LIN {X 0,Y 382.688,Z 736.187,A -85,B 0,C 180,E1 16955.399,E2 16955.399} C_VEL
LIN {X 0,Y 386.297,Z 719.198,A -85,B 0,C 180,E1 16953.634,E2 16953.634} C_VEL
LIN {X 0,Y 389.635,Z 701.414,A -85,B 0,C 180,E1 16952.136,E2 16952.136} C_VEL
LIN {X 0,Y 392.651,Z 682.888,A -85,B 0,C 180,E1 16950.895,E2 16950.895} C_VEL
LIN {X 0,Y 395.335,Z 662.731,A -85,B 0,C 180,E1 16949.855,E2 16949.855} C_VEL
LIN {X 0,Y 397.472,Z 642.044,A -85,B 0,C 180,E1 16949.087,E2 16949.087} C_VEL
LIN {X 0,Y 399.251,Z 615.615,A -85,B 0,C 180,E1 16948.447,E2 16948.447} C_VEL
LIN {X 0,Y 408.41,Z 452.206,A -85,B 0,C 180,E1 16945.014,E2 16945.014} C_VEL
LIN {X 0,Y 404.369,Z 398.592,A -85,B 0,C 180,E1 16942.698,E2 16942.698} C_VEL
LIN {X 0,Y 403.693,Z 388.775,A -85,B 0,C 180,E1 16942.223,E2 16942.223} C_VEL
LIN {X 0,Y 411.245,Z 343.049,A -85,B 0,C 180,E1 16938.531,E2 16938.531} C_VEL
LIN {X 0,Y 405.242,Z 328.597,A -85,B 0,C 180,E1 16935.6,E2 16935.6} C_VEL
LIN {X 0,Y 399.503,Z 315.936,A -85,B 0,C 180,E1 16932.576,E2 16932.576} C_VEL
LIN {X 0,Y 394.557,Z 306.307,A -85,B 0,C 180,E1 16929.775,E2 16929.775} C_VEL
LIN {X 0,Y 390.908,Z 299.036,A -85,B 0,C 180,E1 16927.347,E2 16927.347} C_VEL
LIN {X 0,Y 387.906,Z 293.83,A -85,B 0,C 180,E1 16925.175,E2 16925.175} C_VEL
LIN {X 0,Y 385.327,Z 289.182,A -85,B 0,C 180,E1 16922.974,E2 16922.974} C_VEL
LIN {X 0,Y 382.942,Z 284.925,A -85,B 0,C 180,E1 16920.436,E2 16920.436} C_VEL
LIN {X 0,Y 382.29,Z 283.961,A -85,B 0,C 180,E1 16919.7,E2 16919.7} C_VEL
LIN {X 0,Y 379.591,Z 279.036,A -85,B 0,C 180,E1 16914.407,E2 16914.407} C_VEL
LIN {X 0,Y 379.173,Z 278.59,A -85,B 0,C 180,E1 16910.59,E2 16910.59} C_VEL
LIN {X 0,Y 379.911,Z 279.467,A -85,B 0,C 180,E1 16907.691,E2 16907.691} C_VEL
LIN {X 0,Y 382.64,Z 284.104,A -85,B 0,C 180,E1 16903.139,E2 16903.139} C_VEL
LIN {X 0,Y 383.425,Z 284.941,A -85,B 0,C 180,E1 16902.392,E2 16902.392} C_VEL
LIN {X 0,Y 385.824,Z 289.277,A -85,B 0,C 180,E1 16899.996,E2 16899.996} C_VEL
LIN {X 0,Y 386.815,Z 290.588,A -85,B 0,C 180,E1 16899.26,E2 16899.26} C_VEL
LIN {X 0,Y 389.166,Z 294.616,A -85,B 0,C 180,E1 16897.491,E2 16897.491} C_VEL
LIN {X 0,Y 393.023,Z 301.294,A -85,B 0,C 180,E1 16895.019,E2 16895.019} C_VEL
LIN {X 0,Y 397.476,Z 309.022,A -85,B 0,C 180,E1 16892.591,E2 16892.591} C_VEL
LIN {X 0,Y 402.971,Z 319.612,A -85,B 0,C 180,E1 16889.92,E2 16889.92} C_VEL
LIN {X 0,Y 408.692,Z 331.236,A -85,B 0,C 180,E1 16887.437,E2 16887.437} C_VEL
LIN {X 0,Y 411.334,Z 336.632,A -85,B 0,C 180,E1 16886.468,E2 16886.468} C_VEL
LIN {X 0,Y 417.132,Z 345.96,A -85,B 0,C 180,E1 16885.268,E2 16885.268} C_VEL
LIN {X 0,Y 417.545,Z 355.442,A -85,B 0,C 180,E1 16884.962,E2 16884.962} C_VEL
LIN {X 0,Y 410.945,Z 542.625,A -85,B 0,C 180,E1 16881.466,E2 16881.466} C_VEL
LIN {X 0,Y 407.268,Z 659.162,A -85,B 0,C 180,E1 16879.351,E2 16879.351} C_VEL
LIN {X 0,Y 405.386,Z 681.756,A -85,B 0,C 180,E1 16878.737,E2 16878.737} C_VEL
LIN {X 0,Y 402.869,Z 703.945,A -85,B 0,C 180,E1 16877.905,E2 16877.905} C_VEL
LIN {X 0,Y 399.919,Z 724.711,A -85,B 0,C 180,E1 16876.887,E2 16876.887} C_VEL
LIN {X 0,Y 396.281,Z 746.248,A -85,B 0,C 180,E1 16875.562,E2 16875.562} C_VEL
LIN {X 0,Y 392.531,Z 766.4,A -85,B 0,C 180,E1 16874.055,E2 16874.055} C_VEL
LIN {X 0,Y 388.456,Z 785.774,A -85,B 0,C 180,E1 16872.303,E2 16872.303} C_VEL
LIN {X 0,Y 384.097,Z 805.442,A -85,B 0,C 180,E1 16870.207,E2 16870.207} C_VEL
LIN {X 0,Y 380.023,Z 823.04,A -85,B 0,C 180,E1 16867.998,E2 16867.998} C_VEL
LIN {X 0,Y 375.819,Z 840.992,A -85,B 0,C 180,E1 16865.353,E2 16865.353} C_VEL
LIN {X 0,Y 372.203,Z 856.686,A -85,B 0,C 180,E1 16862.678,E2 16862.678} C_VEL
LIN {X 0,Y 368.937,Z 871.382,A -85,B 0,C 180,E1 16859.73,E2 16859.73} C_VEL
LIN {X 0,Y 366.041,Z 885.503,A -85,B 0,C 180,E1 16856.437,E2 16856.437} C_VEL
LIN {X 0,Y 363.942,Z 896.95,A -85,B 0,C 180,E1 16853.302,E2 16853.302} C_VEL
LIN {X 0,Y 362.3,Z 907.595,A -85,B 0,C 180,E1 16849.841,E2 16849.841} C_VEL
LIN {X 0,Y 361.331,Z 915.623,A -85,B 0,C 180,E1 16846.723,E2 16846.723} C_VEL
LIN {X 0,Y 360.676,Z 923.062,A -85,B 0,C 180,E1 16843.137,E2 16843.137} C_VEL
LIN {X 0,Y 360.397,Z 928.023,A -85,B 0,C 180,E1 16840.064,E2 16840.064} C_VEL
LIN {X 0,Y 360.333,Z 932.128,A -85,B 0,C 180,E1 16836.531,E2 16836.531} C_VEL
LIN {X 0,Y 360.329,Z 934.234,A -85,B 0,C 180,E1 16833.498,E2 16833.498} C_VEL
LIN {X 0,Y 360.326,Z 935.127,A -85,B 0,C 180,E1 16830.475,E2 16830.475} C_VEL
LIN {X 0,Y 360.322,Z 934.598,A -85,B 0,C 180,E1 16827.135,E2 16827.135} C_VEL
LIN {X 0,Y 360.305,Z 932.768,A -85,B 0,C 180,E1 16824.105,E2 16824.105} C_VEL
LIN {X 0,Y 360.331,Z 929.542,A -85,B 0,C 180,E1 16820.898,E2 16820.898} C_VEL
LIN {X 0,Y 360.586,Z 924.375,A -85,B 0,C 180,E1 16817.435,E2 16817.435} C_VEL
LIN {X 0,Y 361.071,Z 918.244,A -85,B 0,C 180,E1 16814.252,E2 16814.252} C_VEL
LIN {X 0,Y 362.037,Z 909.95,A -85,B 0,C 180,E1 16810.812,E2 16810.812} C_VEL
LIN {X 0,Y 363.482,Z 900.51,A -85,B 0,C 180,E1 16807.558,E2 16807.558} C_VEL
LIN {X 0,Y 365.577,Z 888.949,A -85,B 0,C 180,E1 16804.222,E2 16804.222} C_VEL
LIN {X 0,Y 368.207,Z 876.331,A -85,B 0,C 180,E1 16801.094,E2 16801.094} C_VEL
LIN {X 0,Y 371.344,Z 862.246,A -85,B 0,C 180,E1 16798.146,E2 16798.146} C_VEL
LIN {X 0,Y 375.147,Z 846.088,A -85,B 0,C 180,E1 16795.223,E2 16795.223} C_VEL
LIN {X 0,Y 379.148,Z 829.472,A -85,B 0,C 180,E1 16792.659,E2 16792.659} C_VEL
LIN {X 0,Y 383.39,Z 811.434,A -85,B 0,C 180,E1 16790.285,E2 16790.285} C_VEL
LIN {X 0,Y 387.72,Z 792.747,A -85,B 0,C 180,E1 16788.183,E2 16788.183} C_VEL
LIN {X 0,Y 391.873,Z 773.311,A -85,B 0,C 180,E1 16786.354,E2 16786.354} C_VEL
LIN {X 0,Y 396.014,Z 752.373,A -85,B 0,C 180,E1 16784.697,E2 16784.697} C_VEL
LIN {X 0,Y 399.383,Z 733.203,A -85,B 0,C 180,E1 16783.445,E2 16783.445} C_VEL
LIN {X 0,Y 402.81,Z 710.278,A -85,B 0,C 180,E1 16782.24,E2 16782.24} C_VEL
LIN {X 0,Y 405.545,Z 688.092,A -85,B 0,C 180,E1 16781.334,E2 16781.334} C_VEL
LIN {X 0,Y 407.597,Z 665.402,A -85,B 0,C 180,E1 16780.677,E2 16780.677} C_VEL
LIN {X 0,Y 408.984,Z 634.84,A -85,B 0,C 180,E1 16780.061,E2 16780.061} C_VEL
LIN {X 0,Y 415.34,Z 444.739,A -85,B 0,C 180,E1 16776.571,E2 16776.571} C_VEL
LIN {X 0,Y 418.612,Z 352.233,A -85,B 0,C 180,E1 16774.81,E2 16774.81} C_VEL
LIN {X 0,Y 418.047,Z 346.712,A -85,B 0,C 180,E1 16774.593,E2 16774.593} C_VEL
LIN {X 0,Y 406.732,Z 329.749,A -85,B 0,C 180,E1 16772.405,E2 16772.405} C_VEL
LIN {X 0,Y 397.743,Z 312.998,A -85,B 0,C 180,E1 16769.189,E2 16769.189} C_VEL
LIN {X 0,Y 388.439,Z 296.63,A -85,B 0,C 180,E1 16765.541,E2 16765.541} C_VEL
LIN {X 0,Y 381.638,Z 285.645,A -85,B 0,C 180,E1 16762.652,E2 16762.652} C_VEL
LIN {X 0,Y 378.529,Z 280.582,A -85,B 0,C 180,E1 16761.216,E2 16761.216} C_VEL
LIN {X 0,Y 375.523,Z 275.76,A -85,B 0,C 180,E1 16759.764,E2 16759.764} C_VEL
LIN {X 0,Y 372.969,Z 271.522,A -85,B 0,C 180,E1 16758.442,E2 16758.442} C_VEL
LIN {X 0,Y 369.781,Z 266.966,A -85,B 0,C 180,E1 16756.818,E2 16756.818} C_VEL
LIN {X 0,Y 369.096,Z 265.429,A -85,B 0,C 180,E1 16756.364,E2 16756.364} C_VEL
LIN {X 0,Y 366.486,Z 262.302,A -85,B 0,C 180,E1 16755.022,E2 16755.022} C_VEL
LIN {X 0,Y 365.135,Z 259.526,A -85,B 0,C 180,E1 16754.106,E2 16754.106} C_VEL
LIN {X 0,Y 362.664,Z 256.791,A -85,B 0,C 180,E1 16752.742,E2 16752.742} C_VEL
LIN {X 0,Y 361.846,Z 254.324,A -85,B 0,C 180,E1 16751.88,E2 16751.88} C_VEL
LIN {X 0,Y 361.788,Z 253.955,A -85,B 0,C 180,E1 16749.706,E2 16749.706} C_VEL
LIN {X 0,Y 361.798,Z 253.95,A -85,B 0,C 180,E1 16745.71,E2 16745.71} C_VEL
LIN {X 0,Y 361.799,Z 253.95,A -85,B 0,C 180,E1 16741.584,E2 16741.584} C_VEL
LIN {X 0,Y 361.798,Z 253.959,A -85,B 0,C 180,E1 16737.466,E2 16737.466} C_VEL
LIN {X 0,Y 361.808,Z 253.977,A -85,B 0,C 180,E1 16733.335,E2 16733.335} C_VEL
LIN {X 0,Y 361.798,Z 253.972,A -85,B 0,C 180,E1 16729.169,E2 16729.169} C_VEL
LIN {X 0,Y 361.807,Z 253.951,A -85,B 0,C 180,E1 16725.108,E2 16725.108} C_VEL
LIN {X 0,Y 361.801,Z 253.946,A -85,B 0,C 180,E1 16720.936,E2 16720.936} C_VEL
LIN {X 0,Y 361.808,Z 253.959,A -85,B 0,C 180,E1 16716.896,E2 16716.896} C_VEL
LIN {X 0,Y 361.807,Z 253.98,A -85,B 0,C 180,E1 16712.695,E2 16712.695} C_VEL
LIN {X 0,Y 361.804,Z 253.97,A -85,B 0,C 180,E1 16708.514,E2 16708.514} C_VEL
LIN {X 0,Y 361.798,Z 253.956,A -85,B 0,C 180,E1 16704.331,E2 16704.331} C_VEL
LIN {X 0,Y 361.801,Z 253.949,A -85,B 0,C 180,E1 16700.2,E2 16700.2} C_VEL
LIN {X 0,Y 361.8,Z 253.95,A -85,B 0,C 180,E1 16696.081,E2 16696.081} C_VEL
LIN {X 0,Y 361.802,Z 253.953,A -85,B 0,C 180,E1 16691.975,E2 16691.975} C_VEL
LIN {X 0,Y 361.843,Z 254.237,A -85,B 0,C 180,E1 16690.381,E2 16690.381} C_VEL
LIN {X 0,Y 363.417,Z 257.875,A -85,B 0,C 180,E1 16689.055,E2 16689.055} C_VEL
LIN {X 0,Y 365.534,Z 260.297,A -85,B 0,C 180,E1 16687.896,E2 16687.896} C_VEL
LIN {X 0,Y 367.518,Z 264.005,A -85,B 0,C 180,E1 16686.626,E2 16686.626} C_VEL
LIN {X 0,Y 368.956,Z 265.786,A -85,B 0,C 180,E1 16685.878,E2 16685.878} C_VEL
LIN {X 0,Y 371.04,Z 269.542,A -85,B 0,C 180,E1 16684.653,E2 16684.653} C_VEL
LIN {X 0,Y 372.261,Z 271.21,A -85,B 0,C 180,E1 16684.046,E2 16684.046} C_VEL
LIN {X 0,Y 374.624,Z 275.216,A -85,B 0,C 180,E1 16682.785,E2 16682.785} C_VEL
LIN {X 0,Y 378.879,Z 282.66,A -85,B 0,C 180,E1 16680.62,E2 16680.62} C_VEL
LIN {X 0,Y 383.531,Z 290.759,A -85,B 0,C 180,E1 16678.42,E2 16678.42} C_VEL
LIN {X 0,Y 390.609,Z 304.107,A -85,B 0,C 180,E1 16675.236,E2 16675.236} C_VEL
LIN {X 0,Y 397.071,Z 317.353,A -85,B 0,C 180,E1 16672.464,E2 16672.464} C_VEL
LIN {X 0,Y 403.782,Z 332.36,A -85,B 0,C 180,E1 16669.681,E2 16669.681} C_VEL
LIN {X 0,Y 405.757,Z 337.501,A -85,B 0,C 180,E1 16668.834,E2 16668.834} C_VEL
LIN {X 0,Y 398.051,Z 391.605,A -85,B 0,C 180,E1 16664.549,E2 16664.549} C_VEL
LIN {X 0,Y 397.459,Z 397.862,A -85,B 0,C 180,E1 16664.105,E2 16664.105} C_VEL
LIN {X 0,Y 402.131,Z 451.79,A -85,B 0,C 180,E1 16662.007,E2 16662.007} C_VEL
LIN {X 0,Y 393.972,Z 628.533,A -85,B 0,C 180,E1 16658.434,E2 16658.434} C_VEL
LIN {X 0,Y 392.449,Z 649.279,A -85,B 0,C 180,E1 16657.835,E2 16657.835} C_VEL
LIN {X 0,Y 391.777,Z 656.525,A -85,B 0,C 180,E1 16657.565,E2 16657.565} C_VEL
LIN {X 0,Y 390.077,Z 664.06,A -85,B 0,C 180,E1 16657.353,E2 16657.353} C_VEL
LIN {X 0,Y 383.174,Z 682.726,A -85,B 0,C 180,E1 16656.918,E2 16656.918} C_VEL
LIN {X 0,Y 381.385,Z 689.741,A -85,B 0,C 180,E1 16656.564,E2 16656.564} C_VEL
LIN {X 0,Y 378.3,Z 708.589,A -85,B 0,C 180,E1 16655.157,E2 16655.157} C_VEL
LIN {X 0,Y 375.005,Z 726.153,A -85,B 0,C 180,E1 16653.517,E2 16653.517} C_VEL
LIN {X 0,Y 371.571,Z 742.681,A -85,B 0,C 180,E1 16651.621,E2 16651.621} C_VEL
LIN {X 0,Y 368.244,Z 757.61,A -85,B 0,C 180,E1 16649.535,E2 16649.535} C_VEL
LIN {X 0,Y 364.986,Z 771.54,A -85,B 0,C 180,E1 16647.175,E2 16647.175} C_VEL
LIN {X 0,Y 362.021,Z 783.964,A -85,B 0,C 180,E1 16644.613,E2 16644.613} C_VEL
LIN {X 0,Y 359.452,Z 794.899,A -85,B 0,C 180,E1 16641.846,E2 16641.846} C_VEL
LIN {X 0,Y 357.411,Z 803.86,A -85,B 0,C 180,E1 16639.036,E2 16639.036} C_VEL
LIN {X 0,Y 355.833,Z 811.436,A -85,B 0,C 180,E1 16636.018,E2 16636.018} C_VEL
LIN {X 0,Y 354.721,Z 817.412,A -85,B 0,C 180,E1 16632.848,E2 16632.848} C_VEL
LIN {X 0,Y 354.064,Z 821.587,A -85,B 0,C 180,E1 16629.641,E2 16629.641} C_VEL
LIN {X 0,Y 353.771,Z 823.967,A -85,B 0,C 180,E1 16626.517,E2 16626.517} C_VEL
LIN {X 0,Y 353.745,Z 824.748,A -85,B 0,C 180,E1 16623.272,E2 16623.272} C_VEL
LIN {X 0,Y 353.963,Z 823.882,A -85,B 0,C 180,E1 16620.133,E2 16620.133} C_VEL
LIN {X 0,Y 354.483,Z 821.421,A -85,B 0,C 180,E1 16617.02,E2 16617.02} C_VEL
LIN {X 0,Y 355.382,Z 817.422,A -85,B 0,C 180,E1 16613.986,E2 16613.986} C_VEL
LIN {X 0,Y 356.758,Z 811.625,A -85,B 0,C 180,E1 16610.909,E2 16610.909} C_VEL
LIN {X 0,Y 358.765,Z 803.801,A -85,B 0,C 180,E1 16607.808,E2 16607.808} C_VEL
LIN {X 0,Y 361.316,Z 794.333,A -85,B 0,C 180,E1 16604.881,E2 16604.881} C_VEL
LIN {X 0,Y 364.284,Z 783.463,A -85,B 0,C 180,E1 16602.18,E2 16602.18} C_VEL
LIN {X 0,Y 367.641,Z 771.125,A -85,B 0,C 180,E1 16599.68,E2 16599.68} C_VEL
LIN {X 0,Y 371.24,Z 757.424,A -85,B 0,C 180,E1 16597.393,E2 16597.393} C_VEL
LIN {X 0,Y 375.158,Z 741.609,A -85,B 0,C 180,E1 16595.231,E2 16595.231} C_VEL
LIN {X 0,Y 378.942,Z 725.002,A -85,B 0,C 180,E1 16593.378,E2 16593.378} C_VEL
LIN {X 0,Y 382.663,Z 706.838,A -85,B 0,C 180,E1 16591.738,E2 16591.738} C_VEL
LIN {X 0,Y 385.974,Z 688.136,A -85,B 0,C 180,E1 16590.391,E2 16590.391} C_VEL
LIN {X 0,Y 388.913,Z 668.177,A -85,B 0,C 180,E1 16589.28,E2 16589.28} C_VEL
LIN {X 0,Y 391.268,Z 647.69,A -85,B 0,C 180,E1 16588.442,E2 16588.442} C_VEL
LIN {X 0,Y 392.994,Z 626.19,A -85,B 0,C 180,E1 16587.852,E2 16587.852} C_VEL
LIN {X 0,Y 403.129,Z 453.659,A -85,B 0,C 180,E1 16584.186,E2 16584.186} C_VEL
LIN {X 0,Y 399.359,Z 400.422,A -85,B 0,C 180,E1 16581.845,E2 16581.845} C_VEL
LIN {X 0,Y 398.52,Z 387.636,A -85,B 0,C 180,E1 16581.217,E2 16581.217} C_VEL
LIN {X 0,Y 405.502,Z 347.225,A -85,B 0,C 180,E1 16577.914,E2 16577.914} C_VEL
LIN {X 0,Y 399.966,Z 333.564,A -85,B 0,C 180,E1 16575.069,E2 16575.069} C_VEL
LIN {X 0,Y 394.644,Z 321.669,A -85,B 0,C 180,E1 16572.138,E2 16572.138} C_VEL
LIN {X 0,Y 389.914,Z 312.135,A -85,B 0,C 180,E1 16569.296,E2 16569.296} C_VEL
LIN {X 0,Y 386.341,Z 305.126,A -85,B 0,C 180,E1 16566.837,E2 16566.837} C_VEL
LIN {X 0,Y 383.92,Z 300.595,A -85,B 0,C 180,E1 16564.93,E2 16564.93} C_VEL
LIN {X 0,Y 381.583,Z 296.206,A -85,B 0,C 180,E1 16562.853,E2 16562.853} C_VEL
LIN {X 0,Y 379.28,Z 292.042,A -85,B 0,C 180,E1 16560.302,E2 16560.302} C_VEL
LIN {X 0,Y 378.639,Z 291.04,A -85,B 0,C 180,E1 16559.546,E2 16559.546} C_VEL
LIN {X 0,Y 376.196,Z 286.275,A -85,B 0,C 180,E1 16554.356,E2 16554.356} C_VEL
LIN {X 0,Y 375.815,Z 285.853,A -85,B 0,C 180,E1 16550.66,E2 16550.66} C_VEL
LIN {X 0,Y 376.492,Z 286.609,A -85,B 0,C 180,E1 16547.889,E2 16547.889} C_VEL
LIN {X 0,Y 379.308,Z 291.4,A -85,B 0,C 180,E1 16543.104,E2 16543.104} C_VEL
LIN {X 0,Y 379.969,Z 292.424,A -85,B 0,C 180,E1 16542.385,E2 16542.385} C_VEL
LIN {X 0,Y 382.656,Z 296.799,A -85,B 0,C 180,E1 16539.823,E2 16539.823} C_VEL
LIN {X 0,Y 386.131,Z 302.923,A -85,B 0,C 180,E1 16537.144,E2 16537.144} C_VEL
LIN {X 0,Y 389.061,Z 308.123,A -85,B 0,C 180,E1 16535.235,E2 16535.235} C_VEL
LIN {X 0,Y 393.424,Z 315.935,A -85,B 0,C 180,E1 16532.777,E2 16532.777} C_VEL
LIN {X 0,Y 398.532,Z 325.948,A -85,B 0,C 180,E1 16530.214,E2 16530.214} C_VEL
LIN {X 0,Y 404.028,Z 337.304,A -85,B 0,C 180,E1 16527.771,E2 16527.771} C_VEL
LIN {X 0,Y 412.063,Z 350.006,A -85,B 0,C 180,E1 16525.992,E2 16525.992} C_VEL
LIN {X 0,Y 412.277,Z 356.873,A -85,B 0,C 180,E1 16525.778,E2 16525.778} C_VEL
LIN {X 0,Y 405.196,Z 546.047,A -85,B 0,C 180,E1 16522.205,E2 16522.205} C_VEL
LIN {X 0,Y 401.455,Z 658.643,A -85,B 0,C 180,E1 16520.14,E2 16520.14} C_VEL
LIN {X 0,Y 399.525,Z 681.093,A -85,B 0,C 180,E1 16519.526,E2 16519.526} C_VEL
LIN {X 0,Y 396.954,Z 702.973,A -85,B 0,C 180,E1 16518.705,E2 16518.705} C_VEL
LIN {X 0,Y 393.979,Z 723.237,A -85,B 0,C 180,E1 16517.71,E2 16517.71} C_VEL
LIN {X 0,Y 390.175,Z 744.944,A -85,B 0,C 180,E1 16516.377,E2 16516.377} C_VEL
LIN {X 0,Y 386.094,Z 765.857,A -85,B 0,C 180,E1 16514.8,E2 16514.8} C_VEL
LIN {X 0,Y 381.823,Z 785.265,A -85,B 0,C 180,E1 16513.02,E2 16513.02} C_VEL
LIN {X 0,Y 377.134,Z 805.454,A -85,B 0,C 180,E1 16510.826,E2 16510.826} C_VEL
LIN {X 0,Y 372.713,Z 823.659,A -85,B 0,C 180,E1 16508.487,E2 16508.487} C_VEL
LIN {X 0,Y 368.468,Z 840.841,A -85,B 0,C 180,E1 16505.88,E2 16505.88} C_VEL
LIN {X 0,Y 364.583,Z 856.807,A -85,B 0,C 180,E1 16503.074,E2 16503.074} C_VEL
LIN {X 0,Y 361.194,Z 871.379,A -85,B 0,C 180,E1 16500.067,E2 16500.067} C_VEL
LIN {X 0,Y 358.189,Z 885.306,A -85,B 0,C 180,E1 16496.704,E2 16496.704} C_VEL
LIN {X 0,Y 355.929,Z 897.222,A -85,B 0,C 180,E1 16493.332,E2 16493.332} C_VEL
LIN {X 0,Y 354.338,Z 907.121,A -85,B 0,C 180,E1 16489.962,E2 16489.962} C_VEL
LIN {X 0,Y 353.271,Z 915.827,A -85,B 0,C 180,E1 16486.439,E2 16486.439} C_VEL
LIN {X 0,Y 352.71,Z 922.339,A -85,B 0,C 180,E1 16483.106,E2 16483.106} C_VEL
LIN {X 0,Y 352.438,Z 927.45,A -85,B 0,C 180,E1 16479.799,E2 16479.799} C_VEL
LIN {X 0,Y 352.416,Z 931.153,A -85,B 0,C 180,E1 16476.351,E2 16476.351} C_VEL
LIN {X 0,Y 352.417,Z 933.167,A -85,B 0,C 180,E1 16473.251,E2 16473.251} C_VEL
LIN {X 0,Y 352.426,Z 933.964,A -85,B 0,C 180,E1 16469.836,E2 16469.836} C_VEL
LIN {X 0,Y 352.406,Z 933.164,A -85,B 0,C 180,E1 16466.583,E2 16466.583} C_VEL
LIN {X 0,Y 352.389,Z 931.171,A -85,B 0,C 180,E1 16463.482,E2 16463.482} C_VEL
LIN {X 0,Y 352.428,Z 927.232,A -85,B 0,C 180,E1 16459.868,E2 16459.868} C_VEL
LIN {X 0,Y 352.699,Z 922.401,A -85,B 0,C 180,E1 16456.723,E2 16456.723} C_VEL
LIN {X 0,Y 353.328,Z 915.548,A -85,B 0,C 180,E1 16453.222,E2 16453.222} C_VEL
LIN {X 0,Y 354.392,Z 907.299,A -85,B 0,C 180,E1 16449.865,E2 16449.865} C_VEL
LIN {X 0,Y 356.129,Z 896.907,A -85,B 0,C 180,E1 16446.328,E2 16446.328} C_VEL
LIN {X 0,Y 358.359,Z 885.68,A -85,B 0,C 180,E1 16443.127,E2 16443.127} C_VEL
LIN {X 0,Y 361.444,Z 871.823,A -85,B 0,C 180,E1 16439.769,E2 16439.769} C_VEL
LIN {X 0,Y 365.071,Z 856.773,A -85,B 0,C 180,E1 16436.651,E2 16436.651} C_VEL
LIN {X 0,Y 369.093,Z 840.617,A -85,B 0,C 180,E1 16433.83,E2 16433.83} C_VEL
LIN {X 0,Y 373.575,Z 822.695,A -85,B 0,C 180,E1 16431.156,E2 16431.156} C_VEL
LIN {X 0,Y 378.141,Z 804.314,A -85,B 0,C 180,E1 16428.821,E2 16428.821} C_VEL
LIN {X 0,Y 382.576,Z 785.189,A -85,B 0,C 180,E1 16426.784,E2 16426.784} C_VEL
LIN {X 0,Y 386.861,Z 765.624,A -85,B 0,C 180,E1 16425.018,E2 16425.018} C_VEL
LIN {X 0,Y 390.768,Z 745.695,A -85,B 0,C 180,E1 16423.527,E2 16423.527} C_VEL
LIN {X 0,Y 394.634,Z 723.464,A -85,B 0,C 180,E1 16422.176,E2 16422.176} C_VEL
LIN {X 0,Y 397.727,Z 702.475,A -85,B 0,C 180,E1 16421.154,E2 16421.154} C_VEL
LIN {X 0,Y 400.204,Z 680.919,A -85,B 0,C 180,E1 16420.364,E2 16420.364} C_VEL
LIN {X 0,Y 402.111,Z 658.063,A -85,B 0,C 180,E1 16419.752,E2 16419.752} C_VEL
LIN {X 0,Y 409.524,Z 448.97,A -85,B 0,C 180,E1 16415.862,E2 16415.862} C_VEL
LIN {X 0,Y 413.094,Z 353.38,A -85,B 0,C 180,E1 16414.021,E2 16414.021} C_VEL
LIN {X 0,Y 412.732,Z 350.864,A -85,B 0,C 180,E1 16413.903,E2 16413.903} C_VEL
LIN {X 0,Y 400.038,Z 332.096,A -85,B 0,C 180,E1 16411.408,E2 16411.408} C_VEL
LIN {X 0,Y 391.985,Z 317.207,A -85,B 0,C 180,E1 16408.489,E2 16408.489} C_VEL
LIN {X 0,Y 383.66,Z 302.559,A -85,B 0,C 180,E1 16405.138,E2 16405.138} C_VEL
LIN {X 0,Y 377.067,Z 291.755,A -85,B 0,C 180,E1 16402.264,E2 16402.264} C_VEL
LIN {X 0,Y 373.99,Z 286.758,A -85,B 0,C 180,E1 16400.829,E2 16400.829} C_VEL
LIN {X 0,Y 371.353,Z 282.381,A -85,B 0,C 180,E1 16399.504,E2 16399.504} C_VEL
LIN {X 0,Y 367.881,Z 276.964,A -85,B 0,C 180,E1 16397.723,E2 16397.723} C_VEL
LIN {X 0,Y 365.437,Z 273.053,A -85,B 0,C 180,E1 16396.369,E2 16396.369} C_VEL
LIN {X 0,Y 364.319,Z 271.513,A -85,B 0,C 180,E1 16395.766,E2 16395.766} C_VEL
LIN {X 0,Y 361.953,Z 267.903,A -85,B 0,C 180,E1 16394.396,E2 16394.396} C_VEL
LIN {X 0,Y 361.313,Z 266.486,A -85,B 0,C 180,E1 16393.932,E2 16393.932} C_VEL
LIN {X 0,Y 358.607,Z 263.337,A -85,B 0,C 180,E1 16392.398,E2 16392.398} C_VEL
LIN {X 0,Y 357.402,Z 260.703,A -85,B 0,C 180,E1 16391.457,E2 16391.457} C_VEL
LIN {X 0,Y 354.849,Z 257.921,A -85,B 0,C 180,E1 16389.898,E2 16389.898} C_VEL
LIN {X 0,Y 353.871,Z 255.276,A -85,B 0,C 180,E1 16388.777,E2 16388.777} C_VEL
LIN {X 0,Y 353.856,Z 254.939,A -85,B 0,C 180,E1 16385.676,E2 16385.676} C_VEL
LIN {X 0,Y 353.853,Z 254.938,A -85,B 0,C 180,E1 16381.458,E2 16381.458} C_VEL
LIN {X 0,Y 353.856,Z 254.946,A -85,B 0,C 180,E1 16377.409,E2 16377.409} C_VEL
LIN {X 0,Y 353.858,Z 254.962,A -85,B 0,C 180,E1 16373.185,E2 16373.185} C_VEL
LIN {X 0,Y 353.85,Z 254.966,A -85,B 0,C 180,E1 16368.923,E2 16368.923} C_VEL
LIN {X 0,Y 353.851,Z 254.945,A -85,B 0,C 180,E1 16364.765,E2 16364.765} C_VEL
LIN {X 0,Y 353.852,Z 254.935,A -85,B 0,C 180,E1 16360.696,E2 16360.696} C_VEL
LIN {X 0,Y 353.855,Z 254.942,A -85,B 0,C 180,E1 16356.522,E2 16356.522} C_VEL
LIN {X 0,Y 353.858,Z 254.963,A -85,B 0,C 180,E1 16352.394,E2 16352.394} C_VEL
LIN {X 0,Y 353.86,Z 254.964,A -85,B 0,C 180,E1 16348.268,E2 16348.268} C_VEL
LIN {X 0,Y 353.857,Z 254.948,A -85,B 0,C 180,E1 16344.005,E2 16344.005} C_VEL
LIN {X 0,Y 353.857,Z 254.941,A -85,B 0,C 180,E1 16339.723,E2 16339.723} C_VEL
LIN {X 0,Y 353.86,Z 254.938,A -85,B 0,C 180,E1 16335.515,E2 16335.515} C_VEL
LIN {X 0,Y 353.907,Z 255.258,A -85,B 0,C 180,E1 16333.357,E2 16333.357} C_VEL
LIN {X 0,Y 355.515,Z 258.902,A -85,B 0,C 180,E1 16331.803,E2 16331.803} C_VEL
LIN {X 0,Y 357.682,Z 261.181,A -85,B 0,C 180,E1 16330.507,E2 16330.507} C_VEL
LIN {X 0,Y 359.243,Z 264.517,A -85,B 0,C 180,E1 16329.311,E2 16329.311} C_VEL
LIN {X 0,Y 361.241,Z 266.855,A -85,B 0,C 180,E1 16328.182,E2 16328.182} C_VEL
LIN {X 0,Y 363.371,Z 270.753,A -85,B 0,C 180,E1 16326.803,E2 16326.803} C_VEL
LIN {X 0,Y 364.633,Z 272.426,A -85,B 0,C 180,E1 16326.127,E2 16326.127} C_VEL
LIN {X 0,Y 367.156,Z 276.625,A -85,B 0,C 180,E1 16324.674,E2 16324.674} C_VEL
LIN {X 0,Y 371.11,Z 283.453,A -85,B 0,C 180,E1 16322.512,E2 16322.512} C_VEL
LIN {X 0,Y 374.333,Z 289.087,A -85,B 0,C 180,E1 16320.855,E2 16320.855} C_VEL
LIN {X 0,Y 379.138,Z 297.713,A -85,B 0,C 180,E1 16318.513,E2 16318.513} C_VEL
LIN {X 0,Y 385.611,Z 310.022,A -85,B 0,C 180,E1 16315.535,E2 16315.535} C_VEL
LIN {X 0,Y 392.171,Z 323.682,A -85,B 0,C 180,E1 16312.643,E2 16312.643} C_VEL
LIN {X 0,Y 398.885,Z 339.087,A -85,B 0,C 180,E1 16309.78,E2 16309.78} C_VEL
LIN {X 0,Y 399.624,Z 341.553,A -85,B 0,C 180,E1 16309.398,E2 16309.398} C_VEL
LIN {X 0,Y 391.665,Z 396.092,A -85,B 0,C 180,E1 16305.057,E2 16305.057} C_VEL
LIN {X 0,Y 396.352,Z 452.83,A -85,B 0,C 180,E1 16302.79,E2 16302.79} C_VEL
LIN {X 0,Y 387.846,Z 629.005,A -85,B 0,C 180,E1 16299.185,E2 16299.185} C_VEL
LIN {X 0,Y 386.239,Z 649.943,A -85,B 0,C 180,E1 16298.571,E2 16298.571} C_VEL
LIN {X 0,Y 384.129,Z 669.563,A -85,B 0,C 180,E1 16297.731,E2 16297.731} C_VEL
LIN {X 0,Y 381.468,Z 689.178,A -85,B 0,C 180,E1 16296.602,E2 16296.602} C_VEL
LIN {X 0,Y 381.385,Z 689.741,A -85,B 0,C 180,E1 16296.564,E2 16296.564} C_VEL
LIN {X 0,Y 379.504,Z 696.886,A -85,B 0,C 180,E1 16296.166,E2 16296.166} C_VEL
LIN {X 0,Y 371.617,Z 714.596,A -85,B 0,C 180,E1 16295.314,E2 16295.314} C_VEL
LIN {X 0,Y 369.553,Z 721.101,A -85,B 0,C 180,E1 16294.798,E2 16294.798} C_VEL
LIN {X 0,Y 366.03,Z 737.881,A -85,B 0,C 180,E1 16292.977,E2 16292.977} C_VEL
LIN {X 0,Y 362.404,Z 753.765,A -85,B 0,C 180,E1 16290.871,E2 16290.871} C_VEL
LIN {X 0,Y 358.948,Z 768.045,A -85,B 0,C 180,E1 16288.565,E2 16288.565} C_VEL
LIN {X 0,Y 355.643,Z 781.249,A -85,B 0,C 180,E1 16285.971,E2 16285.971} C_VEL
LIN {X 0,Y 352.741,Z 792.871,A -85,B 0,C 180,E1 16283.164,E2 16283.164} C_VEL
LIN {X 0,Y 350.284,Z 802.924,A -85,B 0,C 180,E1 16280.14,E2 16280.14} C_VEL
LIN {X 0,Y 348.449,Z 810.966,A -85,B 0,C 180,E1 16277.069,E2 16277.069} C_VEL
LIN {X 0,Y 347.178,Z 817.198,A -85,B 0,C 180,E1 16273.952,E2 16273.952} C_VEL
LIN {X 0,Y 346.336,Z 821.944,A -85,B 0,C 180,E1 16270.612,E2 16270.612} C_VEL
LIN {X 0,Y 345.931,Z 824.775,A -85,B 0,C 180,E1 16267.395,E2 16267.395} C_VEL
LIN {X 0,Y 345.831,Z 825.996,A -85,B 0,C 180,E1 16264.045,E2 16264.045} C_VEL
LIN {X 0,Y 346.014,Z 825.5,A -85,B 0,C 180,E1 16260.769,E2 16260.769} C_VEL
LIN {X 0,Y 346.482,Z 823.372,A -85,B 0,C 180,E1 16257.54,E2 16257.54} C_VEL
LIN {X 0,Y 347.338,Z 819.742,A -85,B 0,C 180,E1 16254.448,E2 16254.448} C_VEL
LIN {X 0,Y 348.714,Z 814.267,A -85,B 0,C 180,E1 16251.25,E2 16251.25} C_VEL
LIN {X 0,Y 350.653,Z 807.093,A -85,B 0,C 180,E1 16248.149,E2 16248.149} C_VEL
LIN {X 0,Y 353.175,Z 798.246,A -85,B 0,C 180,E1 16245.179,E2 16245.179} C_VEL
LIN {X 0,Y 356.215,Z 787.715,A -85,B 0,C 180,E1 16242.349,E2 16242.349} C_VEL
LIN {X 0,Y 359.784,Z 775.379,A -85,B 0,C 180,E1 16239.668,E2 16239.668} C_VEL
LIN {X 0,Y 363.634,Z 761.594,A -85,B 0,C 180,E1 16237.222,E2 16237.222} C_VEL
LIN {X 0,Y 367.647,Z 746.427,A -85,B 0,C 180,E1 16235.017,E2 16235.017} C_VEL
LIN {X 0,Y 371.652,Z 730.08,A -85,B 0,C 180,E1 16233.071,E2 16233.071} C_VEL
LIN {X 0,Y 375.436,Z 713.02,A -85,B 0,C 180,E1 16231.418,E2 16231.418} C_VEL
LIN {X 0,Y 379.075,Z 694.205,A -85,B 0,C 180,E1 16229.954,E2 16229.954} C_VEL
LIN {X 0,Y 382.247,Z 674.711,A -85,B 0,C 180,E1 16228.769,E2 16228.769} C_VEL
LIN {X 0,Y 384.908,Z 654.367,A -85,B 0,C 180,E1 16227.842,E2 16227.842} C_VEL
LIN {X 0,Y 386.9,Z 633.572,A -85,B 0,C 180,E1 16227.182,E2 16227.182} C_VEL
LIN {X 0,Y 395.966,Z 487.939,A -85,B 0,C 180,E1 16224.028,E2 16224.028} C_VEL
LIN {X 0,Y 397.9,Z 454.373,A -85,B 0,C 180,E1 16223.304,E2 16223.304} C_VEL
LIN {X 0,Y 394.448,Z 401.366,A -85,B 0,C 180,E1 16220.921,E2 16220.921} C_VEL
LIN {X 0,Y 393.451,Z 387.038,A -85,B 0,C 180,E1 16220.218,E2 16220.218} C_VEL
LIN {X 0,Y 399.844,Z 351.358,A -85,B 0,C 180,E1 16217.274,E2 16217.274} C_VEL
LIN {X 0,Y 394.488,Z 337.965,A -85,B 0,C 180,E1 16214.381,E2 16214.381} C_VEL
LIN {X 0,Y 389.361,Z 326.398,A -85,B 0,C 180,E1 16211.404,E2 16211.404} C_VEL
LIN {X 0,Y 384.706,Z 316.569,A -85,B 0,C 180,E1 16208.368,E2 16208.368} C_VEL
LIN {X 0,Y 381.849,Z 311.188,A -85,B 0,C 180,E1 16206.313,E2 16206.313} C_VEL
LIN {X 0,Y 379.944,Z 307.357,A -85,B 0,C 180,E1 16204.679,E2 16204.679} C_VEL
LIN {X 0,Y 377.691,Z 303.05,A -85,B 0,C 180,E1 16202.579,E2 16202.579} C_VEL
LIN {X 0,Y 375.149,Z 298.246,A -85,B 0,C 180,E1 16199.541,E2 16199.541} C_VEL
LIN {X 0,Y 372.767,Z 293.436,A -85,B 0,C 180,E1 16194.149,E2 16194.149} C_VEL
LIN {X 0,Y 372.502,Z 293.132,A -85,B 0,C 180,E1 16190.42,E2 16190.42} C_VEL
LIN {X 0,Y 373.162,Z 293.993,A -85,B 0,C 180,E1 16187.779,E2 16187.779} C_VEL
LIN {X 0,Y 375.889,Z 298.628,A -85,B 0,C 180,E1 16183.145,E2 16183.145} C_VEL
LIN {X 0,Y 379.363,Z 304.627,A -85,B 0,C 180,E1 16179.641,E2 16179.641} C_VEL
LIN {X 0,Y 382.247,Z 309.742,A -85,B 0,C 180,E1 16177.386,E2 16177.386} C_VEL
LIN {X 0,Y 385.348,Z 315.403,A -85,B 0,C 180,E1 16175.307,E2 16175.307} C_VEL
LIN {X 0,Y 389.266,Z 322.597,A -85,B 0,C 180,E1 16173.032,E2 16173.032} C_VEL
LIN {X 0,Y 394.406,Z 332.864,A -85,B 0,C 180,E1 16170.373,E2 16170.373} C_VEL
LIN {X 0,Y 397.669,Z 339.47,A -85,B 0,C 180,E1 16168.931,E2 16168.931} C_VEL
LIN {X 0,Y 406.206,Z 352.661,A -85,B 0,C 180,E1 16166.94,E2 16166.94} C_VEL
LIN {X 0,Y 407.151,Z 354.626,A -85,B 0,C 180,E1 16166.716,E2 16166.716} C_VEL
LIN {X 0,Y 402.032,Z 482.053,A -85,B 0,C 180,E1 16164.236,E2 16164.236} C_VEL
LIN {X 0,Y 395.703,Z 658.631,A -85,B 0,C 180,E1 16160.943,E2 16160.943} C_VEL
LIN {X 0,Y 393.715,Z 680.888,A -85,B 0,C 180,E1 16160.328,E2 16160.328} C_VEL
LIN {X 0,Y 391.025,Z 702.799,A -85,B 0,C 180,E1 16159.497,E2 16159.497} C_VEL
LIN {X 0,Y 387.921,Z 723.056,A -85,B 0,C 180,E1 16158.491,E2 16158.491} C_VEL
LIN {X 0,Y 383.967,Z 744.621,A -85,B 0,C 180,E1 16157.149,E2 16157.149} C_VEL
LIN {X 0,Y 379.847,Z 764.836,A -85,B 0,C 180,E1 16155.612,E2 16155.612} C_VEL
LIN {X 0,Y 375.308,Z 784.58,A -85,B 0,C 180,E1 16153.782,E2 16153.782} C_VEL
LIN {X 0,Y 370.486,Z 804.427,A -85,B 0,C 180,E1 16151.595,E2 16151.595} C_VEL
LIN {X 0,Y 366.026,Z 821.916,A -85,B 0,C 180,E1 16149.324,E2 16149.324} C_VEL
LIN {X 0,Y 361.522,Z 839.225,A -85,B 0,C 180,E1 16146.673,E2 16146.673} C_VEL
LIN {X 0,Y 357.417,Z 855.293,A -85,B 0,C 180,E1 16143.814,E2 16143.814} C_VEL
LIN {X 0,Y 353.813,Z 869.85,A -85,B 0,C 180,E1 16140.761,E2 16140.761} C_VEL
LIN {X 0,Y 350.614,Z 883.837,A -85,B 0,C 180,E1 16137.329,E2 16137.329} C_VEL
LIN {X 0,Y 348.309,Z 895.223,A -85,B 0,C 180,E1 16134.054,E2 16134.054} C_VEL
LIN {X 0,Y 346.584,Z 905.287,A -85,B 0,C 180,E1 16130.605,E2 16130.605} C_VEL
LIN {X 0,Y 345.466,Z 913.719,A -85,B 0,C 180,E1 16127.168,E2 16127.168} C_VEL
LIN {X 0,Y 344.804,Z 920.745,A -85,B 0,C 180,E1 16123.583,E2 16123.583} C_VEL
LIN {X 0,Y 344.53,Z 925.706,A -85,B 0,C 180,E1 16120.364,E2 16120.364} C_VEL
LIN {X 0,Y 344.483,Z 929.775,A -85,B 0,C 180,E1 16116.665,E2 16116.665} C_VEL
LIN {X 0,Y 344.505,Z 931.861,A -85,B 0,C 180,E1 16113.492,E2 16113.492} C_VEL
LIN {X 0,Y 344.518,Z 932.748,A -85,B 0,C 180,E1 16110.165,E2 16110.165} C_VEL
LIN {X 0,Y 344.493,Z 932.026,A -85,B 0,C 180,E1 16106.671,E2 16106.671} C_VEL
LIN {X 0,Y 344.464,Z 930.08,A -85,B 0,C 180,E1 16103.498,E2 16103.498} C_VEL
LIN {X 0,Y 344.474,Z 926.45,A -85,B 0,C 180,E1 16099.969,E2 16099.969} C_VEL
LIN {X 0,Y 344.729,Z 921.71,A -85,B 0,C 180,E1 16096.752,E2 16096.752} C_VEL
LIN {X 0,Y 345.35,Z 915.021,A -85,B 0,C 180,E1 16093.169,E2 16093.169} C_VEL
LIN {X 0,Y 346.502,Z 906.435,A -85,B 0,C 180,E1 16089.563,E2 16089.563} C_VEL
LIN {X 0,Y 348.217,Z 896.655,A -85,B 0,C 180,E1 16086.116,E2 16086.116} C_VEL
LIN {X 0,Y 350.521,Z 885.505,A -85,B 0,C 180,E1 16082.844,E2 16082.844} C_VEL
LIN {X 0,Y 353.721,Z 871.845,A -85,B 0,C 180,E1 16079.414,E2 16079.414} C_VEL
LIN {X 0,Y 357.101,Z 858.331,A -85,B 0,C 180,E1 16076.523,E2 16076.523} C_VEL
LIN {X 0,Y 361.303,Z 842.257,A -85,B 0,C 180,E1 16073.586,E2 16073.586} C_VEL
LIN {X 0,Y 365.8,Z 825.266,A -85,B 0,C 180,E1 16070.921,E2 16070.921} C_VEL
LIN {X 0,Y 370.345,Z 807.591,A -85,B 0,C 180,E1 16068.588,E2 16068.588} C_VEL
LIN {X 0,Y 375.26,Z 787.682,A -85,B 0,C 180,E1 16066.361,E2 16066.361} C_VEL
LIN {X 0,Y 379.633,Z 768.736,A -85,B 0,C 180,E1 16064.58,E2 16064.58} C_VEL
LIN {X 0,Y 383.929,Z 747.95,A -85,B 0,C 180,E1 16062.961,E2 16062.961} C_VEL
LIN {X 0,Y 387.85,Z 726.889,A -85,B 0,C 180,E1 16061.615,E2 16061.615} C_VEL
LIN {X 0,Y 391.129,Z 705.746,A -85,B 0,C 180,E1 16060.546,E2 16060.546} C_VEL
LIN {X 0,Y 394.018,Z 682.633,A -85,B 0,C 180,E1 16059.652,E2 16059.652} C_VEL
LIN {X 0,Y 396.078,Z 659.988,A -85,B 0,C 180,E1 16059.019,E2 16059.019} C_VEL
LIN {X 0,Y 398.54,Z 593.387,A -85,B 0,C 180,E1 16057.763,E2 16057.763} C_VEL
LIN {X 0,Y 405.847,Z 401.805,A -85,B 0,C 180,E1 16054.149,E2 16054.149} C_VEL
LIN {X 0,Y 407.612,Z 355.236,A -85,B 0,C 180,E1 16053.232,E2 16053.232} C_VEL
LIN {X 0,Y 394.847,Z 336.372,A -85,B 0,C 180,E1 16050.639,E2 16050.639} C_VEL
LIN {X 0,Y 391.608,Z 331.434,A -85,B 0,C 180,E1 16049.86,E2 16049.86} C_VEL
LIN {X 0,Y 383.76,Z 317.095,A -85,B 0,C 180,E1 16046.791,E2 16046.791} C_VEL
LIN {X 0,Y 376.426,Z 304.191,A -85,B 0,C 180,E1 16043.646,E2 16043.646} C_VEL
LIN {X 0,Y 369.793,Z 293.374,A -85,B 0,C 180,E1 16040.579,E2 16040.579} C_VEL
LIN {X 0,Y 366.864,Z 288.6,A -85,B 0,C 180,E1 16039.09,E2 16039.09} C_VEL
LIN {X 0,Y 363.722,Z 283.575,A -85,B 0,C 180,E1 16037.436,E2 16037.436} C_VEL
LIN {X 0,Y 360.476,Z 278.458,A -85,B 0,C 180,E1 16035.608,E2 16035.608} C_VEL
LIN {X 0,Y 357.875,Z 274.48,A -85,B 0,C 180,E1 16034.068,E2 16034.068} C_VEL
LIN {X 0,Y 357.187,Z 273.198,A -85,B 0,C 180,E1 16033.6,E2 16033.6} C_VEL
LIN {X 0,Y 354.556,Z 269.879,A -85,B 0,C 180,E1 16032.046,E2 16032.046} C_VEL
LIN {X 0,Y 353.582,Z 267.663,A -85,B 0,C 180,E1 16031.252,E2 16031.252} C_VEL
LIN {X 0,Y 350.871,Z 264.481,A -85,B 0,C 180,E1 16029.514,E2 16029.514} C_VEL
LIN {X 0,Y 349.586,Z 261.772,A -85,B 0,C 180,E1 16028.388,E2 16028.388} C_VEL
LIN {X 0,Y 346.831,Z 258.813,A -85,B 0,C 180,E1 16026.456,E2 16026.456} C_VEL
LIN {X 0,Y 345.949,Z 256.304,A -85,B 0,C 180,E1 16025.224,E2 16025.224} C_VEL
LIN {X 0,Y 345.891,Z 255.948,A -85,B 0,C 180,E1 16022.817,E2 16022.817} C_VEL
LIN {X 0,Y 345.898,Z 255.961,A -85,B 0,C 180,E1 16018.51,E2 16018.51} C_VEL
LIN {X 0,Y 345.906,Z 255.95,A -85,B 0,C 180,E1 16014.194,E2 16014.194} C_VEL
LIN {X 0,Y 345.911,Z 255.931,A -85,B 0,C 180,E1 16010.013,E2 16010.013} C_VEL
LIN {X 0,Y 345.924,Z 255.922,A -85,B 0,C 180,E1 16005.778,E2 16005.778} C_VEL
LIN {X 0,Y 345.924,Z 255.927,A -85,B 0,C 180,E1 16001.637,E2 16001.637} C_VEL
LIN {X 0,Y 345.935,Z 255.944,A -85,B 0,C 180,E1 15997.394,E2 15997.394} C_VEL
LIN {X 0,Y 345.934,Z 255.959,A -85,B 0,C 180,E1 15993.015,E2 15993.015} C_VEL
LIN {X 0,Y 345.93,Z 255.937,A -85,B 0,C 180,E1 15988.822,E2 15988.822} C_VEL
LIN {X 0,Y 345.922,Z 255.929,A -85,B 0,C 180,E1 15984.482,E2 15984.482} C_VEL
LIN {X 0,Y 345.926,Z 255.924,A -85,B 0,C 180,E1 15980.252,E2 15980.252} C_VEL
LIN {X 0,Y 345.949,Z 256.114,A -85,B 0,C 180,E1 15976.99,E2 15976.99} C_VEL
LIN {X 0,Y 346.319,Z 257.602,A -85,B 0,C 180,E1 15976.141,E2 15976.141} C_VEL
LIN {X 0,Y 348.433,Z 260.823,A -85,B 0,C 180,E1 15974.397,E2 15974.397} C_VEL
LIN {X 0,Y 349.858,Z 262.206,A -85,B 0,C 180,E1 15973.457,E2 15973.457} C_VEL
LIN {X 0,Y 351.654,Z 265.874,A -85,B 0,C 180,E1 15971.928,E2 15971.928} C_VEL
LIN {X 0,Y 353.564,Z 268.076,A -85,B 0,C 180,E1 15970.723,E2 15970.723} C_VEL
LIN {X 0,Y 355.611,Z 271.845,A -85,B 0,C 180,E1 15969.246,E2 15969.246} C_VEL
LIN {X 0,Y 357.011,Z 273.514,A -85,B 0,C 180,E1 15968.445,E2 15968.445} C_VEL
LIN {X 0,Y 359.307,Z 277.584,A -85,B 0,C 180,E1 15966.948,E2 15966.948} C_VEL
LIN {X 0,Y 360.415,Z 279.284,A -85,B 0,C 180,E1 15966.304,E2 15966.304} C_VEL
LIN {X 0,Y 363.63,Z 284.728,A -85,B 0,C 180,E1 15964.424,E2 15964.424} C_VEL
LIN {X 0,Y 366.821,Z 290.272,A -85,B 0,C 180,E1 15962.664,E2 15962.664} C_VEL
LIN {X 0,Y 371.525,Z 298.426,A -85,B 0,C 180,E1 15960.246,E2 15960.246} C_VEL
LIN {X 0,Y 378.609,Z 311.856,A -85,B 0,C 180,E1 15956.798,E2 15956.798} C_VEL
LIN {X 0,Y 385.399,Z 325.863,A -85,B 0,C 180,E1 15953.682,E2 15953.682} C_VEL
LIN {X 0,Y 392.195,Z 341.358,A -85,B 0,C 180,E1 15950.673,E2 15950.673} C_VEL
LIN {X 0,Y 393.613,Z 345.144,A -85,B 0,C 180,E1 15950.018,E2 15950.018} C_VEL
LIN {X 0,Y 385.994,Z 395.6,A -85,B 0,C 180,E1 15945.972,E2 15945.972} C_VEL
LIN {X 0,Y 390.636,Z 453.932,A -85,B 0,C 180,E1 15943.595,E2 15943.595} C_VEL
LIN {X 0,Y 381.797,Z 629.239,A -85,B 0,C 180,E1 15939.964,E2 15939.964} C_VEL
LIN {X 0,Y 380.127,Z 650.208,A -85,B 0,C 180,E1 15939.344,E2 15939.344} C_VEL
LIN {X 0,Y 377.903,Z 670.101,A -85,B 0,C 180,E1 15938.484,E2 15938.484} C_VEL
LIN {X 0,Y 375.155,Z 689.57,A -85,B 0,C 180,E1 15937.351,E2 15937.351} C_VEL
LIN {X 0,Y 371.927,Z 708.631,A -85,B 0,C 180,E1 15935.924,E2 15935.924} C_VEL
LIN {X 0,Y 369.553,Z 721.101,A -85,B 0,C 180,E1 15934.798,E2 15934.798} C_VEL
LIN {X 0,Y 367.455,Z 727.672,A -85,B 0,C 180,E1 15934.24,E2 15934.24} C_VEL
LIN {X 0,Y 359.378,Z 743.005,A -85,B 0,C 180,E1 15933.009,E2 15933.009} C_VEL
LIN {X 0,Y 356.902,Z 748.982,A -85,B 0,C 180,E1 15932.324,E2 15932.324} C_VEL
LIN {X 0,Y 356.677,Z 749.796,A -85,B 0,C 180,E1 15932.211,E2 15932.211} C_VEL
LIN {X 0,Y 353.097,Z 764.172,A -85,B 0,C 180,E1 15930.002,E2 15930.002} C_VEL
LIN {X 0,Y 349.654,Z 777.396,A -85,B 0,C 180,E1 15927.543,E2 15927.543} C_VEL
LIN {X 0,Y 346.529,Z 789.221,A -85,B 0,C 180,E1 15924.87,E2 15924.87} C_VEL
LIN {X 0,Y 343.812,Z 799.634,A -85,B 0,C 180,E1 15921.978,E2 15921.978} C_VEL
LIN {X 0,Y 341.674,Z 808.163,A -85,B 0,C 180,E1 15919.037,E2 15919.037} C_VEL
LIN {X 0,Y 340.023,Z 815.322,A -85,B 0,C 180,E1 15915.875,E2 15915.875} C_VEL
LIN {X 0,Y 338.859,Z 820.998,A -85,B 0,C 180,E1 15912.486,E2 15912.486} C_VEL
LIN {X 0,Y 338.189,Z 824.843,A -85,B 0,C 180,E1 15909.041,E2 15909.041} C_VEL
LIN {X 0,Y 337.941,Z 826.856,A -85,B 0,C 180,E1 15905.679,E2 15905.679} C_VEL
LIN {X 0,Y 337.993,Z 827.18,A -85,B 0,C 180,E1 15902.189,E2 15902.189} C_VEL
LIN {X 0,Y 338.348,Z 825.812,A -85,B 0,C 180,E1 15898.862,E2 15898.862} C_VEL
LIN {X 0,Y 339.111,Z 822.749,A -85,B 0,C 180,E1 15895.523,E2 15895.523} C_VEL
LIN {X 0,Y 340.382,Z 817.938,A -85,B 0,C 180,E1 15892.2,E2 15892.2} C_VEL
LIN {X 0,Y 342.12,Z 811.728,A -85,B 0,C 180,E1 15889.11,E2 15889.11} C_VEL
LIN {X 0,Y 344.53,Z 803.681,A -85,B 0,C 180,E1 15886.03,E2 15886.03} C_VEL
LIN {X 0,Y 347.315,Z 794.555,A -85,B 0,C 180,E1 15883.247,E2 15883.247} C_VEL
LIN {X 0,Y 350.794,Z 783.235,A -85,B 0,C 180,E1 15880.449,E2 15880.449} C_VEL
LIN {X 0,Y 354.814,Z 769.908,A -85,B 0,C 180,E1 15877.777,E2 15877.777} C_VEL
LIN {X 0,Y 358.982,Z 755.407,A -85,B 0,C 180,E1 15875.403,E2 15875.403} C_VEL
LIN {X 0,Y 363.142,Z 739.895,A -85,B 0,C 180,E1 15873.321,E2 15873.321} C_VEL
LIN {X 0,Y 367.363,Z 722.771,A -85,B 0,C 180,E1 15871.451,E2 15871.451} C_VEL
LIN {X 0,Y 371.256,Z 704.906,A -85,B 0,C 180,E1 15869.869,E2 15869.869} C_VEL
LIN {X 0,Y 374.79,Z 686.16,A -85,B 0,C 180,E1 15868.551,E2 15868.551} C_VEL
LIN {X 0,Y 377.788,Z 666.862,A -85,B 0,C 180,E1 15867.497,E2 15867.497} C_VEL
LIN {X 0,Y 380.211,Z 647.003,A -85,B 0,C 180,E1 15866.698,E2 15866.698} C_VEL
LIN {X 0,Y 382.03,Z 625.57,A -85,B 0,C 180,E1 15866.114,E2 15866.114} C_VEL
LIN {X 0,Y 392.866,Z 456.376,A -85,B 0,C 180,E1 15862.451,E2 15862.451} C_VEL
LIN {X 0,Y 389.701,Z 403.264,A -85,B 0,C 180,E1 15860.02,E2 15860.02} C_VEL
LIN {X 0,Y 388.656,Z 385.274,A -85,B 0,C 180,E1 15859.108,E2 15859.108} C_VEL
LIN {X 0,Y 394.286,Z 355.767,A -85,B 0,C 180,E1 15856.651,E2 15856.651} C_VEL
LIN {X 0,Y 389.323,Z 343.018,A -85,B 0,C 180,E1 15853.818,E2 15853.818} C_VEL
LIN {X 0,Y 384.206,Z 331.071,A -85,B 0,C 180,E1 15850.647,E2 15850.647} C_VEL
LIN {X 0,Y 379.728,Z 321.767,A -85,B 0,C 180,E1 15847.565,E2 15847.565} C_VEL
LIN {X 0,Y 377.839,Z 317.929,A -85,B 0,C 180,E1 15846.076,E2 15846.076} C_VEL
LIN {X 0,Y 375.976,Z 314.116,A -85,B 0,C 180,E1 15844.423,E2 15844.423} C_VEL
LIN {X 0,Y 373.833,Z 309.9,A -85,B 0,C 180,E1 15842.299,E2 15842.299} C_VEL
LIN {X 0,Y 371.515,Z 305.33,A -85,B 0,C 180,E1 15839.383,E2 15839.383} C_VEL
LIN {X 0,Y 369.371,Z 300.671,A -85,B 0,C 180,E1 15834.095,E2 15834.095} C_VEL
LIN {X 0,Y 369.166,Z 300.405,A -85,B 0,C 180,E1 15830.332,E2 15830.332} C_VEL
LIN {X 0,Y 369.781,Z 301.259,A -85,B 0,C 180,E1 15827.824,E2 15827.824} C_VEL
LIN {X 0,Y 372.354,Z 305.76,A -85,B 0,C 180,E1 15823.302,E2 15823.302} C_VEL
LIN {X 0,Y 375.601,Z 311.456,A -85,B 0,C 180,E1 15819.915,E2 15819.915} C_VEL
LIN {X 0,Y 378.567,Z 316.981,A -85,B 0,C 180,E1 15817.482,E2 15817.482} C_VEL
LIN {X 0,Y 381.417,Z 322.226,A -85,B 0,C 180,E1 15815.532,E2 15815.532} C_VEL
LIN {X 0,Y 385.339,Z 329.744,A -85,B 0,C 180,E1 15813.161,E2 15813.161} C_VEL
LIN {X 0,Y 390.444,Z 340.091,A -85,B 0,C 180,E1 15810.464,E2 15810.464} C_VEL
LIN {X 0,Y 399.708,Z 354.183,A -85,B 0,C 180,E1 15808.1,E2 15808.1} C_VEL
LIN {X 0,Y 402.187,Z 358.507,A -85,B 0,C 180,E1 15807.51,E2 15807.51} C_VEL
LIN {X 0,Y 394.378,Z 543.023,A -85,B 0,C 180,E1 15803.944,E2 15803.944} C_VEL
LIN {X 0,Y 390.088,Z 658.061,A -85,B 0,C 180,E1 15801.785,E2 15801.785} C_VEL
LIN {X 0,Y 388.028,Z 680.359,A -85,B 0,C 180,E1 15801.165,E2 15801.165} C_VEL
LIN {X 0,Y 385.173,Z 702.643,A -85,B 0,C 180,E1 15800.313,E2 15800.313} C_VEL
LIN {X 0,Y 382.061,Z 722.229,A -85,B 0,C 180,E1 15799.335,E2 15799.335} C_VEL
LIN {X 0,Y 377.975,Z 743.734,A -85,B 0,C 180,E1 15797.99,E2 15797.99} C_VEL
LIN {X 0,Y 373.733,Z 763.625,A -85,B 0,C 180,E1 15796.467,E2 15796.467} C_VEL
LIN {X 0,Y 368.899,Z 783.791,A -85,B 0,C 180,E1 15794.584,E2 15794.584} C_VEL
LIN {X 0,Y 363.74,Z 804.052,A -85,B 0,C 180,E1 15792.316,E2 15792.316} C_VEL
LIN {X 0,Y 358.955,Z 821.973,A -85,B 0,C 180,E1 15789.942,E2 15789.942} C_VEL
LIN {X 0,Y 354.263,Z 839.05,A -85,B 0,C 180,E1 15787.259,E2 15787.259} C_VEL
LIN {X 0,Y 349.864,Z 855.378,A -85,B 0,C 180,E1 15784.261,E2 15784.261} C_VEL
LIN {X 0,Y 346.109,Z 869.871,A -85,B 0,C 180,E1 15781.136,E2 15781.136} C_VEL
LIN {X 0,Y 342.934,Z 883.018,A -85,B 0,C 180,E1 15777.805,E2 15777.805} C_VEL
LIN {X 0,Y 340.406,Z 894.934,A -85,B 0,C 180,E1 15774.279,E2 15774.279} C_VEL
LIN {X 0,Y 338.631,Z 904.826,A -85,B 0,C 180,E1 15770.75,E2 15770.75} C_VEL
LIN {X 0,Y 337.449,Z 913.513,A -85,B 0,C 180,E1 15767.056,E2 15767.056} C_VEL
LIN {X 0,Y 336.837,Z 920.026,A -85,B 0,C 180,E1 15763.56,E2 15763.56} C_VEL
LIN {X 0,Y 336.565,Z 925.139,A -85,B 0,C 180,E1 15760.093,E2 15760.093} C_VEL
LIN {X 0,Y 336.565,Z 928.798,A -85,B 0,C 180,E1 15756.48,E2 15756.48} C_VEL
LIN {X 0,Y 336.593,Z 930.714,A -85,B 0,C 180,E1 15753.404,E2 15753.404} C_VEL
LIN {X 0,Y 336.617,Z 931.55,A -85,B 0,C 180,E1 15749.998,E2 15749.998} C_VEL
LIN {X 0,Y 336.58,Z 930.769,A -85,B 0,C 180,E1 15746.503,E2 15746.503} C_VEL
LIN {X 0,Y 336.533,Z 928.858,A -85,B 0,C 180,E1 15743.344,E2 15743.344} C_VEL
LIN {X 0,Y 336.542,Z 925.208,A -85,B 0,C 180,E1 15739.73,E2 15739.73} C_VEL
LIN {X 0,Y 336.801,Z 920.454,A -85,B 0,C 180,E1 15736.435,E2 15736.435} C_VEL
LIN {X 0,Y 337.462,Z 913.735,A -85,B 0,C 180,E1 15732.764,E2 15732.764} C_VEL
LIN {X 0,Y 338.693,Z 905.096,A -85,B 0,C 180,E1 15729.07,E2 15729.07} C_VEL
LIN {X 0,Y 340.649,Z 894.697,A -85,B 0,C 180,E1 15725.366,E2 15725.366} C_VEL
LIN {X 0,Y 343.158,Z 883.346,A -85,B 0,C 180,E1 15721.988,E2 15721.988} C_VEL
LIN {X 0,Y 346.571,Z 869.562,A -85,B 0,C 180,E1 15718.519,E2 15718.519} C_VEL
LIN {X 0,Y 350.461,Z 855.072,A -85,B 0,C 180,E1 15715.405,E2 15715.405} C_VEL
LIN {X 0,Y 354.822,Z 839.061,A -85,B 0,C 180,E1 15712.505,E2 15712.505} C_VEL
LIN {X 0,Y 359.759,Z 821.17,A -85,B 0,C 180,E1 15709.745,E2 15709.745} C_VEL
LIN {X 0,Y 364.478,Z 803.626,A -85,B 0,C 180,E1 15707.45,E2 15707.45} C_VEL
LIN {X 0,Y 369.254,Z 784.709,A -85,B 0,C 180,E1 15705.368,E2 15705.368} C_VEL
LIN {X 0,Y 373.898,Z 765.245,A -85,B 0,C 180,E1 15703.555,E2 15703.555} C_VEL
LIN {X 0,Y 378.17,Z 745.141,A -85,B 0,C 180,E1 15702.015,E2 15702.015} C_VEL
LIN {X 0,Y 382.362,Z 722.721,A -85,B 0,C 180,E1 15700.627,E2 15700.627} C_VEL
LIN {X 0,Y 385.71,Z 701.444,A -85,B 0,C 180,E1 15699.577,E2 15699.577} C_VEL
LIN {X 0,Y 388.338,Z 679.959,A -85,B 0,C 180,E1 15698.784,E2 15698.784} C_VEL
LIN {X 0,Y 390.334,Z 657.13,A -85,B 0,C 180,E1 15698.167,E2 15698.167} C_VEL
LIN {X 0,Y 398.397,Z 449.524,A -85,B 0,C 180,E1 15694.231,E2 15694.231} C_VEL
LIN {X 0,Y 402.105,Z 359.079,A -85,B 0,C 180,E1 15692.465,E2 15692.465} C_VEL
LIN {X 0,Y 390.466,Z 341.719,A -85,B 0,C 180,E1 15690.02,E2 15690.02} C_VEL
LIN {X 0,Y 384.328,Z 332.888,A -85,B 0,C 180,E1 15688.6,E2 15688.6} C_VEL
LIN {X 0,Y 376.43,Z 318.386,A -85,B 0,C 180,E1 15685.318,E2 15685.318} C_VEL
LIN {X 0,Y 368.998,Z 305.541,A -85,B 0,C 180,E1 15681.959,E2 15681.959} C_VEL
LIN {X 0,Y 362.991,Z 295.598,A -85,B 0,C 180,E1 15678.968,E2 15678.968} C_VEL
LIN {X 0,Y 359.277,Z 289.807,A -85,B 0,C 180,E1 15676.991,E2 15676.991} C_VEL
LIN {X 0,Y 356.325,Z 285.076,A -85,B 0,C 180,E1 15675.294,E2 15675.294} C_VEL
LIN {X 0,Y 353.804,Z 281.052,A -85,B 0,C 180,E1 15673.733,E2 15673.733} C_VEL
LIN {X 0,Y 352.762,Z 279.6,A -85,B 0,C 180,E1 15673.106,E2 15673.106} C_VEL
LIN {X 0,Y 350.323,Z 275.987,A -85,B 0,C 180,E1 15671.525,E2 15671.525} C_VEL
LIN {X 0,Y 349.491,Z 274.39,A -85,B 0,C 180,E1 15670.884,E2 15670.884} C_VEL
LIN {X 0,Y 346.875,Z 271.015,A -85,B 0,C 180,E1 15669.122,E2 15669.122} C_VEL
LIN {X 0,Y 345.784,Z 268.733,A -85,B 0,C 180,E1 15668.146,E2 15668.146} C_VEL
LIN {X 0,Y 343.102,Z 265.707,A -85,B 0,C 180,E1 15666.19,E2 15666.19} C_VEL
LIN {X 0,Y 341.847,Z 262.946,A -85,B 0,C 180,E1 15664.866,E2 15664.866} C_VEL
LIN {X 0,Y 338.893,Z 259.801,A -85,B 0,C 180,E1 15662.368,E2 15662.368} C_VEL
LIN {X 0,Y 338.002,Z 257.26,A -85,B 0,C 180,E1 15660.848,E2 15660.848} C_VEL
LIN {X 0,Y 337.983,Z 256.928,A -85,B 0,C 180,E1 15657.797,E2 15657.797} C_VEL
LIN {X 0,Y 337.993,Z 256.94,A -85,B 0,C 180,E1 15653.376,E2 15653.376} C_VEL
LIN {X 0,Y 337.978,Z 256.936,A -85,B 0,C 180,E1 15649.087,E2 15649.087} C_VEL
LIN {X 0,Y 337.972,Z 256.921,A -85,B 0,C 180,E1 15644.735,E2 15644.735} C_VEL
LIN {X 0,Y 337.97,Z 256.912,A -85,B 0,C 180,E1 15640.471,E2 15640.471} C_VEL
LIN {X 0,Y 337.972,Z 256.915,A -85,B 0,C 180,E1 15636.276,E2 15636.276} C_VEL
LIN {X 0,Y 337.977,Z 256.927,A -85,B 0,C 180,E1 15631.942,E2 15631.942} C_VEL
LIN {X 0,Y 337.986,Z 256.945,A -85,B 0,C 180,E1 15627.627,E2 15627.627} C_VEL
LIN {X 0,Y 337.988,Z 256.938,A -85,B 0,C 180,E1 15623.294,E2 15623.294} C_VEL
LIN {X 0,Y 338.036,Z 257.242,A -85,B 0,C 180,E1 15621.072,E2 15621.072} C_VEL
LIN {X 0,Y 339.932,Z 261.242,A -85,B 0,C 180,E1 15618.564,E2 15618.564} C_VEL
LIN {X 0,Y 342.068,Z 263.377,A -85,B 0,C 180,E1 15616.846,E2 15616.846} C_VEL
LIN {X 0,Y 343.901,Z 267.035,A -85,B 0,C 180,E1 15615.051,E2 15615.051} C_VEL
LIN {X 0,Y 345.837,Z 269.04,A -85,B 0,C 180,E1 15613.709,E2 15613.709} C_VEL
LIN {X 0,Y 347.781,Z 272.835,A -85,B 0,C 180,E1 15612.058,E2 15612.058} C_VEL
LIN {X 0,Y 349.377,Z 274.6,A -85,B 0,C 180,E1 15611.055,E2 15611.055} C_VEL
LIN {X 0,Y 351.375,Z 278.419,A -85,B 0,C 180,E1 15609.545,E2 15609.545} C_VEL
LIN {X 0,Y 352.831,Z 280.279,A -85,B 0,C 180,E1 15608.675,E2 15608.675} C_VEL
LIN {X 0,Y 355.462,Z 284.657,A -85,B 0,C 180,E1 15606.982,E2 15606.982} C_VEL
LIN {X 0,Y 359.425,Z 291.602,A -85,B 0,C 180,E1 15604.573,E2 15604.573} C_VEL
LIN {X 0,Y 364.379,Z 300.104,A -85,B 0,C 180,E1 15601.855,E2 15601.855} C_VEL
LIN {X 0,Y 371.281,Z 313.093,A -85,B 0,C 180,E1 15598.286,E2 15598.286} C_VEL
LIN {X 0,Y 377.781,Z 326.267,A -85,B 0,C 180,E1 15595.158,E2 15595.158} C_VEL
LIN {X 0,Y 384.788,Z 341.931,A -85,B 0,C 180,E1 15591.931,E2 15591.931} C_VEL
LIN {X 0,Y 387.567,Z 349.168,A -85,B 0,C 180,E1 15590.62,E2 15590.62} C_VEL
LIN {X 0,Y 380.412,Z 394.847,A -85,B 0,C 180,E1 15586.929,E2 15586.929} C_VEL
LIN {X 0,Y 385.001,Z 454.943,A -85,B 0,C 180,E1 15584.424,E2 15584.424} C_VEL
LIN {X 0,Y 375.822,Z 629.462,A -85,B 0,C 180,E1 15580.768,E2 15580.768} C_VEL
LIN {X 0,Y 374.097,Z 650.347,A -85,B 0,C 180,E1 15580.147,E2 15580.147} C_VEL
LIN {X 0,Y 371.714,Z 670.86,A -85,B 0,C 180,E1 15579.25,E2 15579.25} C_VEL
LIN {X 0,Y 368.855,Z 690.29,A -85,B 0,C 180,E1 15578.105,E2 15578.105} C_VEL
LIN {X 0,Y 365.533,Z 709.135,A -85,B 0,C 180,E1 15576.677,E2 15576.677} C_VEL
LIN {X 0,Y 361.932,Z 726.835,A -85,B 0,C 180,E1 15575,E2 15575} C_VEL
LIN {X 0,Y 358.151,Z 743.596,A -85,B 0,C 180,E1 15573.042,E2 15573.042} C_VEL
LIN {X 0,Y 356.677,Z 749.796,A -85,B 0,C 180,E1 15572.211,E2 15572.211} C_VEL
LIN {X 0,Y 354.419,Z 755.683,A -85,B 0,C 180,E1 15571.463,E2 15571.463} C_VEL
LIN {X 0,Y 345.61,Z 770.102,A -85,B 0,C 180,E1 15569.662,E2 15569.662} C_VEL
LIN {X 0,Y 343.376,Z 775.165,A -85,B 0,C 180,E1 15568.783,E2 15568.783} C_VEL
LIN {X 0,Y 339.993,Z 787.31,A -85,B 0,C 180,E1 15566.123,E2 15566.123} C_VEL
LIN {X 0,Y 337.129,Z 797.655,A -85,B 0,C 180,E1 15563.36,E2 15563.36} C_VEL
LIN {X 0,Y 334.545,Z 807.224,A -85,B 0,C 180,E1 15560.193,E2 15560.193} C_VEL
LIN {X 0,Y 332.6,Z 814.982,A -85,B 0,C 180,E1 15556.902,E2 15556.902} C_VEL
LIN {X 0,Y 331.255,Z 820.959,A -85,B 0,C 180,E1 15553.519,E2 15553.519} C_VEL
LIN {X 0,Y 330.453,Z 825.064,A -85,B 0,C 180,E1 15550.193,E2 15550.193} C_VEL
LIN {X 0,Y 330.077,Z 827.566,A -85,B 0,C 180,E1 15546.812,E2 15546.812} C_VEL
LIN {X 0,Y 330.028,Z 828.465,A -85,B 0,C 180,E1 15543.556,E2 15543.556} C_VEL
LIN {X 0,Y 330.266,Z 827.865,A -85,B 0,C 180,E1 15540.234,E2 15540.234} C_VEL
LIN {X 0,Y 330.875,Z 825.614,A -85,B 0,C 180,E1 15536.828,E2 15536.828} C_VEL
LIN {X 0,Y 331.993,Z 821.595,A -85,B 0,C 180,E1 15533.396,E2 15533.396} C_VEL
LIN {X 0,Y 333.761,Z 815.601,A -85,B 0,C 180,E1 15529.906,E2 15529.906} C_VEL
LIN {X 0,Y 336.171,Z 807.925,A -85,B 0,C 180,E1 15526.606,E2 15526.606} C_VEL
LIN {X 0,Y 339.163,Z 798.691,A -85,B 0,C 180,E1 15523.517,E2 15523.517} C_VEL
LIN {X 0,Y 342.738,Z 787.731,A -85,B 0,C 180,E1 15520.582,E2 15520.582} C_VEL
LIN {X 0,Y 346.829,Z 775.004,A -85,B 0,C 180,E1 15517.827,E2 15517.827} C_VEL
LIN {X 0,Y 351.242,Z 760.647,A -85,B 0,C 180,E1 15515.3,E2 15515.3} C_VEL
LIN {X 0,Y 355.795,Z 744.873,A -85,B 0,C 180,E1 15513.036,E2 15513.036} C_VEL
LIN {X 0,Y 360.218,Z 728.132,A -85,B 0,C 180,E1 15511.082,E2 15511.082} C_VEL
LIN {X 0,Y 364.381,Z 710.487,A -85,B 0,C 180,E1 15509.417,E2 15509.417} C_VEL
LIN {X 0,Y 368.134,Z 692.078,A -85,B 0,C 180,E1 15508.025,E2 15508.025} C_VEL
LIN {X 0,Y 371.25,Z 673.991,A -85,B 0,C 180,E1 15506.948,E2 15506.948} C_VEL
LIN {X 0,Y 374.024,Z 653.991,A -85,B 0,C 180,E1 15506.045,E2 15506.045} C_VEL
LIN {X 0,Y 376.156,Z 632.859,A -85,B 0,C 180,E1 15505.383,E2 15505.383} C_VEL
LIN {X 0,Y 386.712,Z 476.291,A -85,B 0,C 180,E1 15501.948,E2 15501.948} C_VEL
LIN {X 0,Y 387.872,Z 456.953,A -85,B 0,C 180,E1 15501.511,E2 15501.511} C_VEL
LIN {X 0,Y 385.043,Z 404.728,A -85,B 0,C 180,E1 15499.071,E2 15499.071} C_VEL
LIN {X 0,Y 383.96,Z 384.184,A -85,B 0,C 180,E1 15498.012,E2 15498.012} C_VEL
LIN {X 0,Y 388.748,Z 360.011,A -85,B 0,C 180,E1 15495.973,E2 15495.973} C_VEL
LIN {X 0,Y 383.979,Z 347.516,A -85,B 0,C 180,E1 15493.093,E2 15493.093} C_VEL
LIN {X 0,Y 379.513,Z 336.896,A -85,B 0,C 180,E1 15490.166,E2 15490.166} C_VEL
LIN {X 0,Y 375.633,Z 328.485,A -85,B 0,C 180,E1 15487.34,E2 15487.34} C_VEL
LIN {X 0,Y 373.652,Z 324.333,A -85,B 0,C 180,E1 15485.681,E2 15485.681} C_VEL
LIN {X 0,Y 372.013,Z 320.873,A -85,B 0,C 180,E1 15484.161,E2 15484.161} C_VEL
LIN {X 0,Y 369.989,Z 316.741,A -85,B 0,C 180,E1 15482.013,E2 15482.013} C_VEL
LIN {X 0,Y 367.923,Z 312.431,A -85,B 0,C 180,E1 15479.221,E2 15479.221} C_VEL
LIN {X 0,Y 365.954,Z 307.881,A -85,B 0,C 180,E1 15473.977,E2 15473.977} C_VEL
LIN {X 0,Y 365.818,Z 307.675,A -85,B 0,C 180,E1 15470.243,E2 15470.243} C_VEL
LIN {X 0,Y 366.355,Z 308.387,A -85,B 0,C 180,E1 15468.028,E2 15468.028} C_VEL
LIN {X 0,Y 369.198,Z 313.539,A -85,B 0,C 180,E1 15462.993,E2 15462.993} C_VEL
LIN {X 0,Y 371.978,Z 318.661,A -85,B 0,C 180,E1 15460.039,E2 15460.039} C_VEL
LIN {X 0,Y 374.719,Z 323.805,A -85,B 0,C 180,E1 15457.734,E2 15457.734} C_VEL
LIN {X 0,Y 377.821,Z 329.646,A -85,B 0,C 180,E1 15455.549,E2 15455.549} C_VEL
LIN {X 0,Y 382.483,Z 338.805,A -85,B 0,C 180,E1 15452.718,E2 15452.718} C_VEL
LIN {X 0,Y 384.537,Z 342.843,A -85,B 0,C 180,E1 15451.713,E2 15451.713} C_VEL
LIN {X 0,Y 393.235,Z 355.72,A -85,B 0,C 180,E1 15449.349,E2 15449.349} C_VEL
LIN {X 0,Y 397.163,Z 362.405,A -85,B 0,C 180,E1 15448.351,E2 15448.351} C_VEL
LIN {X 0,Y 389.054,Z 544.062,A -85,B 0,C 180,E1 15444.807,E2 15444.807} C_VEL
LIN {X 0,Y 384.543,Z 657.961,A -85,B 0,C 180,E1 15442.643,E2 15442.643} C_VEL
LIN {X 0,Y 382.422,Z 680.103,A -85,B 0,C 180,E1 15442.022,E2 15442.022} C_VEL
LIN {X 0,Y 379.426,Z 702.513,A -85,B 0,C 180,E1 15441.158,E2 15441.158} C_VEL
LIN {X 0,Y 376.164,Z 722.176,A -85,B 0,C 180,E1 15440.164,E2 15440.164} C_VEL
LIN {X 0,Y 371.893,Z 743.676,A -85,B 0,C 180,E1 15438.799,E2 15438.799} C_VEL
LIN {X 0,Y 367.36,Z 763.973,A -85,B 0,C 180,E1 15437.221,E2 15437.221} C_VEL
LIN {X 0,Y 362.466,Z 783.453,A -85,B 0,C 180,E1 15435.37,E2 15435.37} C_VEL
LIN {X 0,Y 357.106,Z 803.497,A -85,B 0,C 180,E1 15433.089,E2 15433.089} C_VEL
LIN {X 0,Y 352.17,Z 821.199,A -85,B 0,C 180,E1 15430.707,E2 15430.707} C_VEL
LIN {X 0,Y 347.304,Z 837.949,A -85,B 0,C 180,E1 15428.028,E2 15428.028} C_VEL
LIN {X 0,Y 342.813,Z 853.846,A -85,B 0,C 180,E1 15425.067,E2 15425.067} C_VEL
LIN {X 0,Y 339.005,Z 867.591,A -85,B 0,C 180,E1 15422.063,E2 15422.063} C_VEL
LIN {X 0,Y 335.385,Z 881.783,A -85,B 0,C 180,E1 15418.422,E2 15418.422} C_VEL
LIN {X 0,Y 332.712,Z 893.672,A -85,B 0,C 180,E1 15414.829,E2 15414.829} C_VEL
LIN {X 0,Y 330.756,Z 903.911,A -85,B 0,C 180,E1 15411.081,E2 15411.081} C_VEL
LIN {X 0,Y 329.52,Z 912.536,A -85,B 0,C 180,E1 15407.297,E2 15407.297} C_VEL
LIN {X 0,Y 328.891,Z 919.021,A -85,B 0,C 180,E1 15403.715,E2 15403.715} C_VEL
LIN {X 0,Y 328.618,Z 924.297,A -85,B 0,C 180,E1 15399.985,E2 15399.985} C_VEL
LIN {X 0,Y 328.642,Z 927.693,A -85,B 0,C 180,E1 15396.462,E2 15396.462} C_VEL
LIN {X 0,Y 328.683,Z 929.649,A -85,B 0,C 180,E1 15393.137,E2 15393.137} C_VEL
LIN {X 0,Y 328.698,Z 930.294,A -85,B 0,C 180,E1 15389.65,E2 15389.65} C_VEL
LIN {X 0,Y 328.664,Z 929.52,A -85,B 0,C 180,E1 15386.335,E2 15386.335} C_VEL
LIN {X 0,Y 328.596,Z 927.508,A -85,B 0,C 180,E1 15383.007,E2 15383.007} C_VEL
LIN {X 0,Y 328.614,Z 923.735,A -85,B 0,C 180,E1 15379.302,E2 15379.302} C_VEL
LIN {X 0,Y 328.909,Z 918.815,A -85,B 0,C 180,E1 15375.868,E2 15375.868} C_VEL
LIN {X 0,Y 329.68,Z 911.641,A -85,B 0,C 180,E1 15371.978,E2 15371.978} C_VEL
LIN {X 0,Y 330.989,Z 903.311,A -85,B 0,C 180,E1 15368.373,E2 15368.373} C_VEL
LIN {X 0,Y 333.237,Z 892.175,A -85,B 0,C 180,E1 15364.4,E2 15364.4} C_VEL
LIN {X 0,Y 336.149,Z 880.116,A -85,B 0,C 180,E1 15360.802,E2 15360.802} C_VEL
LIN {X 0,Y 339.725,Z 866.495,A -85,B 0,C 180,E1 15357.41,E2 15357.41} C_VEL
LIN {X 0,Y 344.184,Z 850.704,A -85,B 0,C 180,E1 15354.067,E2 15354.067} C_VEL
LIN {X 0,Y 348.722,Z 835.029,A -85,B 0,C 180,E1 15351.25,E2 15351.25} C_VEL
LIN {X 0,Y 353.569,Z 818.044,A -85,B 0,C 180,E1 15348.674,E2 15348.674} C_VEL
LIN {X 0,Y 358.613,Z 799.944,A -85,B 0,C 180,E1 15346.327,E2 15346.327} C_VEL
LIN {X 0,Y 363.423,Z 781.582,A -85,B 0,C 180,E1 15344.329,E2 15344.329} C_VEL
LIN {X 0,Y 368.488,Z 760.636,A -85,B 0,C 180,E1 15342.433,E2 15342.433} C_VEL
LIN {X 0,Y 372.827,Z 740.807,A -85,B 0,C 180,E1 15340.946,E2 15340.946} C_VEL
LIN {X 0,Y 376.753,Z 719.732,A -85,B 0,C 180,E1 15339.678,E2 15339.678} C_VEL
LIN {X 0,Y 380.208,Z 697.738,A -85,B 0,C 180,E1 15338.626,E2 15338.626} C_VEL
LIN {X 0,Y 382.742,Z 677.354,A -85,B 0,C 180,E1 15337.894,E2 15337.894} C_VEL
LIN {X 0,Y 384.71,Z 653.57,A -85,B 0,C 180,E1 15337.277,E2 15337.277} C_VEL
LIN {X 0,Y 392.925,Z 449.553,A -85,B 0,C 180,E1 15333.383,E2 15333.383} C_VEL
LIN {X 0,Y 396.63,Z 362.751,A -85,B 0,C 180,E1 15331.667,E2 15331.667} C_VEL
LIN {X 0,Y 384.302,Z 344.399,A -85,B 0,C 180,E1 15328.985,E2 15328.985} C_VEL
LIN {X 0,Y 377.227,Z 334.429,A -85,B 0,C 180,E1 15327.294,E2 15327.294} C_VEL
LIN {X 0,Y 369.833,Z 321,A -85,B 0,C 180,E1 15324.094,E2 15324.094} C_VEL
LIN {X 0,Y 361.74,Z 307.042,A -85,B 0,C 180,E1 15320.213,E2 15320.213} C_VEL
LIN {X 0,Y 355.731,Z 297.157,A -85,B 0,C 180,E1 15316.997,E2 15316.997} C_VEL
LIN {X 0,Y 352.19,Z 291.683,A -85,B 0,C 180,E1 15314.972,E2 15314.972} C_VEL
LIN {X 0,Y 348.919,Z 286.522,A -85,B 0,C 180,E1 15312.916,E2 15312.916} C_VEL
LIN {X 0,Y 346.301,Z 282.525,A -85,B 0,C 180,E1 15311.154,E2 15311.154} C_VEL
LIN {X 0,Y 345.684,Z 281.333,A -85,B 0,C 180,E1 15310.668,E2 15310.668} C_VEL
LIN {X 0,Y 342.903,Z 277.546,A -85,B 0,C 180,E1 15308.722,E2 15308.722} C_VEL
LIN {X 0,Y 341.993,Z 275.689,A -85,B 0,C 180,E1 15307.899,E2 15307.899} C_VEL
LIN {X 0,Y 339.347,Z 272.584,A -85,B 0,C 180,E1 15305.92,E2 15305.92} C_VEL
LIN {X 0,Y 338.09,Z 269.897,A -85,B 0,C 180,E1 15304.58,E2 15304.58} C_VEL
LIN {X 0,Y 335.225,Z 266.67,A -85,B 0,C 180,E1 15302.052,E2 15302.052} C_VEL
LIN {X 0,Y 333.879,Z 263.854,A -85,B 0,C 180,E1 15300.344,E2 15300.344} C_VEL
LIN {X 0,Y 330.921,Z 260.717,A -85,B 0,C 180,E1 15297.056,E2 15297.056} C_VEL
LIN {X 0,Y 330.071,Z 258.24,A -85,B 0,C 180,E1 15294.961,E2 15294.961} C_VEL
LIN {X 0,Y 330.042,Z 257.897,A -85,B 0,C 180,E1 15291.288,E2 15291.288} C_VEL
LIN {X 0,Y 330.04,Z 257.905,A -85,B 0,C 180,E1 15287.046,E2 15287.046} C_VEL
LIN {X 0,Y 330.036,Z 257.924,A -85,B 0,C 180,E1 15282.73,E2 15282.73} C_VEL
LIN {X 0,Y 330.036,Z 257.935,A -85,B 0,C 180,E1 15278.31,E2 15278.31} C_VEL
LIN {X 0,Y 330.038,Z 257.914,A -85,B 0,C 180,E1 15273.943,E2 15273.943} C_VEL
LIN {X 0,Y 330.047,Z 257.902,A -85,B 0,C 180,E1 15269.609,E2 15269.609} C_VEL
LIN {X 0,Y 330.108,Z 258.3,A -85,B 0,C 180,E1 15266.719,E2 15266.719} C_VEL
LIN {X 0,Y 332.508,Z 262.773,A -85,B 0,C 180,E1 15262.815,E2 15262.815} C_VEL
LIN {X 0,Y 334.235,Z 264.41,A -85,B 0,C 180,E1 15261.06,E2 15261.06} C_VEL
LIN {X 0,Y 336.247,Z 268.303,A -85,B 0,C 180,E1 15258.691,E2 15258.691} C_VEL
LIN {X 0,Y 338.163,Z 270.118,A -85,B 0,C 180,E1 15257.154,E2 15257.154} C_VEL
LIN {X 0,Y 339.924,Z 273.801,A -85,B 0,C 180,E1 15255.333,E2 15255.333} C_VEL
LIN {X 0,Y 341.91,Z 276.103,A -85,B 0,C 180,E1 15253.875,E2 15253.875} C_VEL
LIN {X 0,Y 343.955,Z 279.847,A -85,B 0,C 180,E1 15252.162,E2 15252.162} C_VEL
LIN {X 0,Y 345.413,Z 281.731,A -85,B 0,C 180,E1 15251.184,E2 15251.184} C_VEL
LIN {X 0,Y 347.936,Z 285.929,A -85,B 0,C 180,E1 15249.376,E2 15249.376} C_VEL
LIN {X 0,Y 351.913,Z 292.676,A -85,B 0,C 180,E1 15246.755,E2 15246.755} C_VEL
LIN {X 0,Y 355.005,Z 298.004,A -85,B 0,C 180,E1 15244.873,E2 15244.873} C_VEL
LIN {X 0,Y 359.924,Z 306.664,A -85,B 0,C 180,E1 15242.085,E2 15242.085} C_VEL
LIN {X 0,Y 366.286,Z 318.714,A -85,B 0,C 180,E1 15238.715,E2 15238.715} C_VEL
LIN {X 0,Y 372.969,Z 332.547,A -85,B 0,C 180,E1 15235.39,E2 15235.39} C_VEL
LIN {X 0,Y 379.653,Z 347.857,A -85,B 0,C 180,E1 15232.207,E2 15232.207} C_VEL
LIN {X 0,Y 381.636,Z 352.745,A -85,B 0,C 180,E1 15231.277,E2 15231.277} C_VEL
LIN {X 0,Y 374.909,Z 393.947,A -85,B 0,C 180,E1 15227.917,E2 15227.917} C_VEL
LIN {X 0,Y 379.433,Z 455.96,A -85,B 0,C 180,E1 15225.275,E2 15225.275} C_VEL
LIN {X 0,Y 369.891,Z 630.004,A -85,B 0,C 180,E1 15221.59,E2 15221.59} C_VEL
LIN {X 0,Y 368.065,Z 651.18,A -85,B 0,C 180,E1 15220.949,E2 15220.949} C_VEL
LIN {X 0,Y 365.692,Z 670.881,A -85,B 0,C 180,E1 15220.079,E2 15220.079} C_VEL
LIN {X 0,Y 362.809,Z 689.888,A -85,B 0,C 180,E1 15218.959,E2 15218.959} C_VEL
LIN {X 0,Y 359.522,Z 708.055,A -85,B 0,C 180,E1 15217.593,E2 15217.593} C_VEL
LIN {X 0,Y 355.863,Z 725.555,A -85,B 0,C 180,E1 15215.954,E2 15215.954} C_VEL
LIN {X 0,Y 352.07,Z 741.904,A -85,B 0,C 180,E1 15214.073,E2 15214.073} C_VEL
LIN {X 0,Y 348.291,Z 756.919,A -85,B 0,C 180,E1 15211.976,E2 15211.976} C_VEL
LIN {X 0,Y 344.405,Z 771.458,A -85,B 0,C 180,E1 15209.503,E2 15209.503} C_VEL
LIN {X 0,Y 343.376,Z 775.165,A -85,B 0,C 180,E1 15208.783,E2 15208.783} C_VEL
LIN {X 0,Y 341.166,Z 780.195,A -85,B 0,C 180,E1 15207.862,E2 15207.862} C_VEL
LIN {X 0,Y 332.898,Z 791.788,A -85,B 0,C 180,E1 15205.718,E2 15205.718} C_VEL
LIN {X 0,Y 330.537,Z 796.014,A -85,B 0,C 180,E1 15204.671,E2 15204.671} C_VEL
LIN {X 0,Y 330.344,Z 796.572,A -85,B 0,C 180,E1 15204.508,E2 15204.508} C_VEL
LIN {X 0,Y 327.562,Z 806.264,A -85,B 0,C 180,E1 15201.4,E2 15201.4} C_VEL
LIN {X 0,Y 325.357,Z 814.347,A -85,B 0,C 180,E1 15198.12,E2 15198.12} C_VEL
LIN {X 0,Y 323.81,Z 820.627,A -85,B 0,C 180,E1 15194.786,E2 15194.786} C_VEL
LIN {X 0,Y 322.767,Z 825.441,A -85,B 0,C 180,E1 15191.208,E2 15191.208} C_VEL
LIN {X 0,Y 322.236,Z 828.466,A -85,B 0,C 180,E1 15187.566,E2 15187.566} C_VEL
LIN {X 0,Y 322.116,Z 829.685,A -85,B 0,C 180,E1 15184.047,E2 15184.047} C_VEL
LIN {X 0,Y 322.346,Z 829.235,A -85,B 0,C 180,E1 15180.452,E2 15180.452} C_VEL
LIN {X 0,Y 322.94,Z 827.155,A -85,B 0,C 180,E1 15176.984,E2 15176.984} C_VEL
LIN {X 0,Y 324.007,Z 823.572,A -85,B 0,C 180,E1 15173.649,E2 15173.649} C_VEL
LIN {X 0,Y 325.635,Z 818.339,A -85,B 0,C 180,E1 15170.311,E2 15170.311} C_VEL
LIN {X 0,Y 328.005,Z 811.181,A -85,B 0,C 180,E1 15166.939,E2 15166.939} C_VEL
LIN {X 0,Y 331.006,Z 802.471,A -85,B 0,C 180,E1 15163.766,E2 15163.766} C_VEL
LIN {X 0,Y 334.588,Z 792.102,A -85,B 0,C 180,E1 15160.756,E2 15160.756} C_VEL
LIN {X 0,Y 338.649,Z 780.249,A -85,B 0,C 180,E1 15157.975,E2 15157.975} C_VEL
LIN {X 0,Y 342.973,Z 767.174,A -85,B 0,C 180,E1 15155.459,E2 15155.459} C_VEL
LIN {X 0,Y 347.578,Z 752.419,A -85,B 0,C 180,E1 15153.13,E2 15153.13} C_VEL
LIN {X 0,Y 352.051,Z 736.942,A -85,B 0,C 180,E1 15151.123,E2 15151.123} C_VEL
LIN {X 0,Y 356.569,Z 719.707,A -85,B 0,C 180,E1 15149.304,E2 15149.304} C_VEL
LIN {X 0,Y 360.771,Z 701.397,A -85,B 0,C 180,E1 15147.748,E2 15147.748} C_VEL
LIN {X 0,Y 364.452,Z 682.5,A -85,B 0,C 180,E1 15146.481,E2 15146.481} C_VEL
LIN {X 0,Y 367.571,Z 662.844,A -85,B 0,C 180,E1 15145.471,E2 15145.471} C_VEL
LIN {X 0,Y 370.017,Z 642.799,A -85,B 0,C 180,E1 15144.726,E2 15144.726} C_VEL
LIN {X 0,Y 372.33,Z 613.713,A -85,B 0,C 180,E1 15144.006,E2 15144.006} C_VEL
LIN {X 0,Y 383.052,Z 458.609,A -85,B 0,C 180,E1 15140.592,E2 15140.592} C_VEL
LIN {X 0,Y 380.567,Z 406.663,A -85,B 0,C 180,E1 15138.119,E2 15138.119} C_VEL
LIN {X 0,Y 379.516,Z 382.622,A -85,B 0,C 180,E1 15136.845,E2 15136.845} C_VEL
LIN {X 0,Y 383.273,Z 364.294,A -85,B 0,C 180,E1 15135.276,E2 15135.276} C_VEL
LIN {X 0,Y 378.707,Z 352.087,A -85,B 0,C 180,E1 15132.348,E2 15132.348} C_VEL
LIN {X 0,Y 374.871,Z 342.72,A -85,B 0,C 180,E1 15129.673,E2 15129.673} C_VEL
LIN {X 0,Y 371.376,Z 334.825,A -85,B 0,C 180,E1 15126.958,E2 15126.958} C_VEL
LIN {X 0,Y 368.425,Z 328.179,A -85,B 0,C 180,E1 15124.201,E2 15124.201} C_VEL
LIN {X 0,Y 366.307,Z 323.789,A -85,B 0,C 180,E1 15121.876,E2 15121.876} C_VEL
LIN {X 0,Y 364.335,Z 319.531,A -85,B 0,C 180,E1 15119.056,E2 15119.056} C_VEL
LIN {X 0,Y 362.525,Z 315.083,A -85,B 0,C 180,E1 15113.825,E2 15113.825} C_VEL
LIN {X 0,Y 362.561,Z 315.026,A -85,B 0,C 180,E1 15109.673,E2 15109.673} C_VEL
LIN {X 0,Y 363.012,Z 315.814,A -85,B 0,C 180,E1 15107.891,E2 15107.891} C_VEL
LIN {X 0,Y 365.666,Z 320.711,A -85,B 0,C 180,E1 15103.133,E2 15103.133} C_VEL
LIN {X 0,Y 368.23,Z 325.487,A -85,B 0,C 180,E1 15100.324,E2 15100.324} C_VEL
LIN {X 0,Y 370.886,Z 330.631,A -85,B 0,C 180,E1 15097.992,E2 15097.992} C_VEL
LIN {X 0,Y 374.281,Z 337.12,A -85,B 0,C 180,E1 15095.539,E2 15095.539} C_VEL
LIN {X 0,Y 377.774,Z 344.177,A -85,B 0,C 180,E1 15093.387,E2 15093.387} C_VEL
LIN {X 0,Y 385.222,Z 354.904,A -85,B 0,C 180,E1 15091.133,E2 15091.133} C_VEL
LIN {X 0,Y 392.289,Z 366.169,A -85,B 0,C 180,E1 15089.222,E2 15089.222} C_VEL
LIN {X 0,Y 383.711,Z 547.766,A -85,B 0,C 180,E1 15085.643,E2 15085.643} C_VEL
LIN {X 0,Y 379.139,Z 657.446,A -85,B 0,C 180,E1 15083.539,E2 15083.539} C_VEL
LIN {X 0,Y 376.941,Z 679.621,A -85,B 0,C 180,E1 15082.913,E2 15082.913} C_VEL
LIN {X 0,Y 373.768,Z 702.397,A -85,B 0,C 180,E1 15082.028,E2 15082.028} C_VEL
LIN {X 0,Y 370.361,Z 722.163,A -85,B 0,C 180,E1 15081.021,E2 15081.021} C_VEL
LIN {X 0,Y 366.213,Z 742.273,A -85,B 0,C 180,E1 15079.736,E2 15079.736} C_VEL
LIN {X 0,Y 361.592,Z 762.207,A -85,B 0,C 180,E1 15078.186,E2 15078.186} C_VEL
LIN {X 0,Y 356.371,Z 782.166,A -85,B 0,C 180,E1 15076.284,E2 15076.284} C_VEL
LIN {X 0,Y 350.743,Z 802.288,A -85,B 0,C 180,E1 15073.979,E2 15073.979} C_VEL
LIN {X 0,Y 345.46,Z 820.376,A -85,B 0,C 180,E1 15071.51,E2 15071.51} C_VEL
LIN {X 0,Y 340.276,Z 837.368,A -85,B 0,C 180,E1 15068.744,E2 15068.744} C_VEL
LIN {X 0,Y 335.211,Z 854.328,A -85,B 0,C 180,E1 15065.482,E2 15065.482} C_VEL
LIN {X 0,Y 330.946,Z 869.172,A -85,B 0,C 180,E1 15062.12,E2 15062.12} C_VEL
LIN {X 0,Y 327.488,Z 882.037,A -85,B 0,C 180,E1 15058.64,E2 15058.64} C_VEL
LIN {X 0,Y 324.619,Z 894.22,A -85,B 0,C 180,E1 15054.762,E2 15054.762} C_VEL
LIN {X 0,Y 322.786,Z 903.596,A -85,B 0,C 180,E1 15051.192,E2 15051.192} C_VEL
LIN {X 0,Y 321.508,Z 912.255,A -85,B 0,C 180,E1 15047.182,E2 15047.182} C_VEL
LIN {X 0,Y 320.902,Z 918.604,A -85,B 0,C 180,E1 15043.512,E2 15043.512} C_VEL
LIN {X 0,Y 320.677,Z 923.792,A -85,B 0,C 180,E1 15039.51,E2 15039.51} C_VEL
LIN {X 0,Y 320.727,Z 926.721,A -85,B 0,C 180,E1 15036.262,E2 15036.262} C_VEL
LIN {X 0,Y 320.778,Z 928.711,A -85,B 0,C 180,E1 15032.499,E2 15032.499} C_VEL
LIN {X 0,Y 320.791,Z 929.015,A -85,B 0,C 180,E1 15029.105,E2 15029.105} C_VEL
LIN {X 0,Y 320.74,Z 928.148,A -85,B 0,C 180,E1 15025.887,E2 15025.887} C_VEL
LIN {X 0,Y 320.648,Z 925.717,A -85,B 0,C 180,E1 15022.112,E2 15022.112} C_VEL
LIN {X 0,Y 320.704,Z 921.782,A -85,B 0,C 180,E1 15018.489,E2 15018.489} C_VEL
LIN {X 0,Y 321.067,Z 916.481,A -85,B 0,C 180,E1 15014.834,E2 15014.834} C_VEL
LIN {X 0,Y 321.975,Z 909.149,A -85,B 0,C 180,E1 15010.968,E2 15010.968} C_VEL
LIN {X 0,Y 323.485,Z 900.613,A -85,B 0,C 180,E1 15007.27,E2 15007.27} C_VEL
LIN {X 0,Y 325.762,Z 890.173,A -85,B 0,C 180,E1 15003.572,E2 15003.572} C_VEL
LIN {X 0,Y 328.911,Z 877.923,A -85,B 0,C 180,E1 14999.893,E2 14999.893} C_VEL
LIN {X 0,Y 332.551,Z 864.945,A -85,B 0,C 180,E1 14996.617,E2 14996.617} C_VEL
LIN {X 0,Y 337.137,Z 849.406,A -85,B 0,C 180,E1 14993.291,E2 14993.291} C_VEL
LIN {X 0,Y 342.115,Z 833.083,A -85,B 0,C 180,E1 14990.323,E2 14990.323} C_VEL
LIN {X 0,Y 347.315,Z 815.521,A -85,B 0,C 180,E1 14987.649,E2 14987.649} C_VEL
LIN {X 0,Y 352.826,Z 796.372,A -85,B 0,C 180,E1 14985.203,E2 14985.203} C_VEL
LIN {X 0,Y 357.922,Z 777.636,A -85,B 0,C 180,E1 14983.187,E2 14983.187} C_VEL
LIN {X 0,Y 362.767,Z 757.896,A -85,B 0,C 180,E1 14981.435,E2 14981.435} C_VEL
LIN {X 0,Y 367.314,Z 737.385,A -85,B 0,C 180,E1 14979.924,E2 14979.924} C_VEL
LIN {X 0,Y 371.239,Z 716.785,A -85,B 0,C 180,E1 14978.703,E2 14978.703} C_VEL
LIN {X 0,Y 374.76,Z 694.161,A -85,B 0,C 180,E1 14977.657,E2 14977.657} C_VEL
LIN {X 0,Y 377.487,Z 672.024,A -85,B 0,C 180,E1 14976.896,E2 14976.896} C_VEL
LIN {X 0,Y 379.16,Z 649.638,A -85,B 0,C 180,E1 14976.358,E2 14976.358} C_VEL
LIN {X 0,Y 387.379,Z 453.283,A -85,B 0,C 180,E1 14972.583,E2 14972.583} C_VEL
LIN {X 0,Y 391.294,Z 366.602,A -85,B 0,C 180,E1 14970.862,E2 14970.862} C_VEL
LIN {X 0,Y 379.25,Z 348.76,A -85,B 0,C 180,E1 14968.159,E2 14968.159} C_VEL
LIN {X 0,Y 369.626,Z 335.23,A -85,B 0,C 180,E1 14965.737,E2 14965.737} C_VEL
LIN {X 0,Y 362.699,Z 322.628,A -85,B 0,C 180,E1 14962.531,E2 14962.531} C_VEL
LIN {X 0,Y 356.304,Z 311.793,A -85,B 0,C 180,E1 14959.338,E2 14959.338} C_VEL
LIN {X 0,Y 351.268,Z 303.368,A -85,B 0,C 180,E1 14956.538,E2 14956.538} C_VEL
LIN {X 0,Y 348.069,Z 298.283,A -85,B 0,C 180,E1 14954.643,E2 14954.643} C_VEL
LIN {X 0,Y 345.083,Z 293.445,A -85,B 0,C 180,E1 14952.722,E2 14952.722} C_VEL
LIN {X 0,Y 342.278,Z 289.054,A -85,B 0,C 180,E1 14950.776,E2 14950.776} C_VEL
LIN {X 0,Y 338.773,Z 283.664,A -85,B 0,C 180,E1 14948.145,E2 14948.145} C_VEL
LIN {X 0,Y 337.927,Z 282.419,A -85,B 0,C 180,E1 14947.481,E2 14947.481} C_VEL
LIN {X 0,Y 335.447,Z 279.122,A -85,B 0,C 180,E1 14945.474,E2 14945.474} C_VEL
LIN {X 0,Y 334.531,Z 277.032,A -85,B 0,C 180,E1 14944.458,E2 14944.458} C_VEL
LIN {X 0,Y 331.68,Z 273.817,A -85,B 0,C 180,E1 14941.901,E2 14941.901} C_VEL
LIN {X 0,Y 330.343,Z 270.989,A -85,B 0,C 180,E1 14940.174,E2 14940.174} C_VEL
LIN {X 0,Y 327.443,Z 267.823,A -85,B 0,C 180,E1 14936.85,E2 14936.85} C_VEL
LIN {X 0,Y 326.201,Z 265.079,A -85,B 0,C 180,E1 14934.548,E2 14934.548} C_VEL
LIN {X 0,Y 322.512,Z 260.649,A -85,B 0,C 180,E1 14926.373,E2 14926.373} C_VEL
LIN {X 0,Y 322.201,Z 259.56,A -85,B 0,C 180,E1 14922.482,E2 14922.482} C_VEL
LIN {X 0,Y 322.227,Z 259.656,A -85,B 0,C 180,E1 14918.523,E2 14918.523} C_VEL
LIN {X 0,Y 322.716,Z 261.13,A -85,B 0,C 180,E1 14914.371,E2 14914.371} C_VEL
LIN {X 0,Y 326.461,Z 265.463,A -85,B 0,C 180,E1 14906.735,E2 14906.735} C_VEL
LIN {X 0,Y 328.868,Z 269.841,A -85,B 0,C 180,E1 14902.989,E2 14902.989} C_VEL
LIN {X 0,Y 330.564,Z 271.469,A -85,B 0,C 180,E1 14901.237,E2 14901.237} C_VEL
LIN {X 0,Y 332.682,Z 275.5,A -85,B 0,C 180,E1 14898.71,E2 14898.71} C_VEL
LIN {X 0,Y 334.4,Z 277.344,A -85,B 0,C 180,E1 14897.257,E2 14897.257} C_VEL
LIN {X 0,Y 336.452,Z 281.19,A -85,B 0,C 180,E1 14895.228,E2 14895.228} C_VEL
LIN {X 0,Y 337.816,Z 282.597,A -85,B 0,C 180,E1 14894.254,E2 14894.254} C_VEL
LIN {X 0,Y 340.043,Z 286.755,A -85,B 0,C 180,E1 14892.328,E2 14892.328} C_VEL
LIN {X 0,Y 341.334,Z 288.529,A -85,B 0,C 180,E1 14891.421,E2 14891.421} C_VEL
LIN {X 0,Y 343.938,Z 292.783,A -85,B 0,C 180,E1 14889.544,E2 14889.544} C_VEL
LIN {X 0,Y 347.757,Z 299.521,A -85,B 0,C 180,E1 14886.937,E2 14886.937} C_VEL
LIN {X 0,Y 351.044,Z 305.293,A -85,B 0,C 180,E1 14884.888,E2 14884.888} C_VEL
LIN {X 0,Y 355.482,Z 313.25,A -85,B 0,C 180,E1 14882.305,E2 14882.305} C_VEL
LIN {X 0,Y 361.668,Z 325.216,A -85,B 0,C 180,E1 14878.935,E2 14878.935} C_VEL
LIN {X 0,Y 368.158,Z 338.817,A -85,B 0,C 180,E1 14875.625,E2 14875.625} C_VEL
LIN {X 0,Y 374.95,Z 354.818,A -85,B 0,C 180,E1 14872.285,E2 14872.285} C_VEL
LIN {X 0,Y 375.687,Z 356.713,A -85,B 0,C 180,E1 14871.923,E2 14871.923} C_VEL
LIN {X 0,Y 369.509,Z 393.125,A -85,B 0,C 180,E1 14868.929,E2 14868.929} C_VEL
LIN {X 0,Y 373.941,Z 457.05,A -85,B 0,C 180,E1 14866.15,E2 14866.15} C_VEL
LIN {X 0,Y 364.051,Z 630.322,A -85,B 0,C 180,E1 14862.442,E2 14862.442} C_VEL
LIN {X 0,Y 362.144,Z 651.623,A -85,B 0,C 180,E1 14861.791,E2 14861.791} C_VEL
LIN {X 0,Y 359.529,Z 672.38,A -85,B 0,C 180,E1 14860.858,E2 14860.858} C_VEL
LIN {X 0,Y 356.45,Z 691.681,A -85,B 0,C 180,E1 14859.691,E2 14859.691} C_VEL
LIN {X 0,Y 352.853,Z 710.527,A -85,B 0,C 180,E1 14858.229,E2 14858.229} C_VEL
LIN {X 0,Y 348.924,Z 728.331,A -85,B 0,C 180,E1 14856.501,E2 14856.501} C_VEL
LIN {X 0,Y 344.812,Z 745.093,A -85,B 0,C 180,E1 14854.492,E2 14854.492} C_VEL
LIN {X 0,Y 340.636,Z 760.776,A -85,B 0,C 180,E1 14852.189,E2 14852.189} C_VEL
LIN {X 0,Y 336.661,Z 774.863,A -85,B 0,C 180,E1 14849.661,E2 14849.661} C_VEL
LIN {X 0,Y 332.985,Z 787.46,A -85,B 0,C 180,E1 14846.904,E2 14846.904} C_VEL
LIN {X 0,Y 330.344,Z 796.572,A -85,B 0,C 180,E1 14844.508,E2 14844.508} C_VEL
LIN {X 0,Y 328.275,Z 800.626,A -85,B 0,C 180,E1 14843.4,E2 14843.4} C_VEL
LIN {X 0,Y 320.055,Z 810.258,A -85,B 0,C 180,E1 14840.639,E2 14840.639} C_VEL
LIN {X 0,Y 318.234,Z 813.42,A -85,B 0,C 180,E1 14839.414,E2 14839.414} C_VEL
LIN {X 0,Y 316.367,Z 820.349,A -85,B 0,C 180,E1 14835.918,E2 14835.918} C_VEL
LIN {X 0,Y 315.108,Z 825.602,A -85,B 0,C 180,E1 14832.267,E2 14832.267} C_VEL
LIN {X 0,Y 314.443,Z 828.961,A -85,B 0,C 180,E1 14828.694,E2 14828.694} C_VEL
LIN {X 0,Y 314.203,Z 830.682,A -85,B 0,C 180,E1 14825.082,E2 14825.082} C_VEL
LIN {X 0,Y 314.314,Z 830.832,A -85,B 0,C 180,E1 14821.709,E2 14821.709} C_VEL
LIN {X 0,Y 314.794,Z 829.456,A -85,B 0,C 180,E1 14818.183,E2 14818.183} C_VEL
LIN {X 0,Y 315.82,Z 826.215,A -85,B 0,C 180,E1 14814.451,E2 14814.451} C_VEL
LIN {X 0,Y 317.508,Z 821.141,A -85,B 0,C 180,E1 14810.774,E2 14810.774} C_VEL
LIN {X 0,Y 319.874,Z 814.389,A -85,B 0,C 180,E1 14807.269,E2 14807.269} C_VEL
LIN {X 0,Y 323.039,Z 805.715,A -85,B 0,C 180,E1 14803.852,E2 14803.852} C_VEL
LIN {X 0,Y 326.823,Z 795.391,A -85,B 0,C 180,E1 14800.653,E2 14800.653} C_VEL
LIN {X 0,Y 331.133,Z 783.557,A -85,B 0,C 180,E1 14797.714,E2 14797.714} C_VEL
LIN {X 0,Y 335.977,Z 769.696,A -85,B 0,C 180,E1 14794.931,E2 14794.931} C_VEL
LIN {X 0,Y 341.079,Z 754.179,A -85,B 0,C 180,E1 14792.412,E2 14792.412} C_VEL
LIN {X 0,Y 346.058,Z 737.766,A -85,B 0,C 180,E1 14790.248,E2 14790.248} C_VEL
LIN {X 0,Y 350.725,Z 720.73,A -85,B 0,C 180,E1 14788.429,E2 14788.429} C_VEL
LIN {X 0,Y 355.182,Z 702.099,A -85,B 0,C 180,E1 14786.832,E2 14786.832} C_VEL
LIN {X 0,Y 359.045,Z 683.106,A -85,B 0,C 180,E1 14785.548,E2 14785.548} C_VEL
LIN {X 0,Y 362.296,Z 663.47,A -85,B 0,C 180,E1 14784.531,E2 14784.531} C_VEL
LIN {X 0,Y 364.848,Z 643.428,A -85,B 0,C 180,E1 14783.779,E2 14783.779} C_VEL
LIN {X 0,Y 367.196,Z 615.192,A -85,B 0,C 180,E1 14783.072,E2 14783.072} C_VEL
LIN {X 0,Y 378.353,Z 459.883,A -85,B 0,C 180,E1 14779.629,E2 14779.629} C_VEL
LIN {X 0,Y 376.176,Z 407.915,A -85,B 0,C 180,E1 14777.109,E2 14777.109} C_VEL
LIN {X 0,Y 375.146,Z 381.666,A -85,B 0,C 180,E1 14775.695,E2 14775.695} C_VEL
LIN {X 0,Y 377.898,Z 368.626,A -85,B 0,C 180,E1 14774.557,E2 14774.557} C_VEL
LIN {X 0,Y 373.758,Z 357.222,A -85,B 0,C 180,E1 14771.73,E2 14771.73} C_VEL
LIN {X 0,Y 369.9,Z 347.605,A -85,B 0,C 180,E1 14768.862,E2 14768.862} C_VEL
LIN {X 0,Y 366.401,Z 339.134,A -85,B 0,C 180,E1 14765.794,E2 14765.794} C_VEL
LIN {X 0,Y 363.979,Z 334.111,A -85,B 0,C 180,E1 14763.464,E2 14763.464} C_VEL
LIN {X 0,Y 362.481,Z 330.623,A -85,B 0,C 180,E1 14761.58,E2 14761.58} C_VEL
LIN {X 0,Y 360.751,Z 326.63,A -85,B 0,C 180,E1 14758.888,E2 14758.888} C_VEL
LIN {X 0,Y 359.116,Z 322.315,A -85,B 0,C 180,E1 14753.766,E2 14753.766} C_VEL
LIN {X 0,Y 359.253,Z 322.333,A -85,B 0,C 180,E1 14749.415,E2 14749.415} C_VEL
LIN {X 0,Y 359.662,Z 323.217,A -85,B 0,C 180,E1 14747.802,E2 14747.802} C_VEL
LIN {X 0,Y 362.131,Z 327.82,A -85,B 0,C 180,E1 14743.312,E2 14743.312} C_VEL
LIN {X 0,Y 364.622,Z 332.681,A -85,B 0,C 180,E1 14740.455,E2 14740.455} C_VEL
LIN {X 0,Y 367.066,Z 337.467,A -85,B 0,C 180,E1 14738.251,E2 14738.251} C_VEL
LIN {X 0,Y 370.356,Z 343.946,A -85,B 0,C 180,E1 14735.772,E2 14735.772} C_VEL
LIN {X 0,Y 371.819,Z 346.604,A -85,B 0,C 180,E1 14734.986,E2 14734.986} C_VEL
LIN {X 0,Y 378.6,Z 356.079,A -85,B 0,C 180,E1 14732.728,E2 14732.728} C_VEL
LIN {X 0,Y 386.591,Z 368.519,A -85,B 0,C 180,E1 14730.375,E2 14730.375} C_VEL
LIN {X 0,Y 387.521,Z 370.417,A -85,B 0,C 180,E1 14730.109,E2 14730.109} C_VEL
LIN {X 0,Y 378.699,Z 547.17,A -85,B 0,C 180,E1 14726.593,E2 14726.593} C_VEL
LIN {X 0,Y 373.823,Z 657.299,A -85,B 0,C 180,E1 14724.454,E2 14724.454} C_VEL
LIN {X 0,Y 371.544,Z 679.474,A -85,B 0,C 180,E1 14723.824,E2 14723.824} C_VEL
LIN {X 0,Y 368.301,Z 701.854,A -85,B 0,C 180,E1 14722.95,E2 14722.95} C_VEL
LIN {X 0,Y 364.632,Z 722.273,A -85,B 0,C 180,E1 14721.901,E2 14721.901} C_VEL
LIN {X 0,Y 360.068,Z 743.322,A -85,B 0,C 180,E1 14720.527,E2 14720.527} C_VEL
LIN {X 0,Y 355.264,Z 763.029,A -85,B 0,C 180,E1 14718.958,E2 14718.958} C_VEL
LIN {X 0,Y 350.047,Z 782.096,A -85,B 0,C 180,E1 14717.106,E2 14717.106} C_VEL
LIN {X 0,Y 344.121,Z 802.262,A -85,B 0,C 180,E1 14714.75,E2 14714.75} C_VEL
LIN {X 0,Y 338.544,Z 820.443,A -85,B 0,C 180,E1 14712.211,E2 14712.211} C_VEL
LIN {X 0,Y 333.15,Z 837.294,A -85,B 0,C 180,E1 14709.399,E2 14709.399} C_VEL
LIN {X 0,Y 328.096,Z 853.343,A -85,B 0,C 180,E1 14706.24,E2 14706.24} C_VEL
LIN {X 0,Y 323.602,Z 868.134,A -85,B 0,C 180,E1 14702.815,E2 14702.815} C_VEL
LIN {X 0,Y 319.879,Z 881.249,A -85,B 0,C 180,E1 14699.181,E2 14699.181} C_VEL
LIN {X 0,Y 316.75,Z 893.797,A -85,B 0,C 180,E1 14695.048,E2 14695.048} C_VEL
LIN {X 0,Y 314.782,Z 903.478,A -85,B 0,C 180,E1 14691.227,E2 14691.227} C_VEL
LIN {X 0,Y 313.537,Z 911.637,A -85,B 0,C 180,E1 14687.25,E2 14687.25} C_VEL
LIN {X 0,Y 312.915,Z 918.186,A -85,B 0,C 180,E1 14683.299,E2 14683.299} C_VEL
LIN {X 0,Y 312.738,Z 922.724,A -85,B 0,C 180,E1 14679.568,E2 14679.568} C_VEL
LIN {X 0,Y 312.805,Z 925.623,A -85,B 0,C 180,E1 14676.231,E2 14676.231} C_VEL
LIN {X 0,Y 312.874,Z 927.521,A -85,B 0,C 180,E1 14672.379,E2 14672.379} C_VEL
LIN {X 0,Y 312.885,Z 927.773,A -85,B 0,C 180,E1 14668.899,E2 14668.899} C_VEL
LIN {X 0,Y 312.819,Z 926.912,A -85,B 0,C 180,E1 14665.746,E2 14665.746} C_VEL
LIN {X 0,Y 312.715,Z 924.648,A -85,B 0,C 180,E1 14662.096,E2 14662.096} C_VEL
LIN {X 0,Y 312.76,Z 920.758,A -85,B 0,C 180,E1 14658.379,E2 14658.379} C_VEL
LIN {X 0,Y 313.098,Z 915.775,A -85,B 0,C 180,E1 14654.818,E2 14654.818} C_VEL
LIN {X 0,Y 314.01,Z 908.596,A -85,B 0,C 180,E1 14650.853,E2 14650.853} C_VEL
LIN {X 0,Y 315.563,Z 900.139,A -85,B 0,C 180,E1 14647.061,E2 14647.061} C_VEL
LIN {X 0,Y 317.916,Z 889.87,A -85,B 0,C 180,E1 14643.271,E2 14643.271} C_VEL
LIN {X 0,Y 321.18,Z 877.781,A -85,B 0,C 180,E1 14639.505,E2 14639.505} C_VEL
LIN {X 0,Y 325.19,Z 864.103,A -85,B 0,C 180,E1 14635.971,E2 14635.971} C_VEL
LIN {X 0,Y 330.131,Z 848.194,A -85,B 0,C 180,E1 14632.498,E2 14632.498} C_VEL
LIN {X 0,Y 335.059,Z 832.773,A -85,B 0,C 180,E1 14629.641,E2 14629.641} C_VEL
LIN {X 0,Y 340.439,Z 815.291,A -85,B 0,C 180,E1 14626.932,E2 14626.932} C_VEL
LIN {X 0,Y 346.218,Z 796.076,A -85,B 0,C 180,E1 14624.43,E2 14624.43} C_VEL
LIN {X 0,Y 351.507,Z 777.378,A -85,B 0,C 180,E1 14622.388,E2 14622.388} C_VEL
LIN {X 0,Y 356.448,Z 758.018,A -85,B 0,C 180,E1 14620.642,E2 14620.642} C_VEL
LIN {X 0,Y 361.036,Z 738.168,A -85,B 0,C 180,E1 14619.154,E2 14619.154} C_VEL
LIN {X 0,Y 365.187,Z 717.053,A -85,B 0,C 180,E1 14617.886,E2 14617.886} C_VEL
LIN {X 0,Y 368.91,Z 694.066,A -85,B 0,C 180,E1 14616.809,E2 14616.809} C_VEL
LIN {X 0,Y 371.744,Z 671.901,A -85,B 0,C 180,E1 14616.039,E2 14616.039} C_VEL
LIN {X 0,Y 373.479,Z 649.456,A -85,B 0,C 180,E1 14615.495,E2 14615.495} C_VEL
LIN {X 0,Y 382.201,Z 449.917,A -85,B 0,C 180,E1 14611.625,E2 14611.625} C_VEL
LIN {X 0,Y 385.908,Z 370.387,A -85,B 0,C 180,E1 14610.026,E2 14610.026} C_VEL
LIN {X 0,Y 373.488,Z 351.916,A -85,B 0,C 180,E1 14607.115,E2 14607.115} C_VEL
LIN {X 0,Y 362.536,Z 336.743,A -85,B 0,C 180,E1 14604.264,E2 14604.264} C_VEL
LIN {X 0,Y 355.669,Z 324.436,A -85,B 0,C 180,E1 14600.918,E2 14600.918} C_VEL
LIN {X 0,Y 349.845,Z 314.546,A -85,B 0,C 180,E1 14597.807,E2 14597.807} C_VEL
LIN {X 0,Y 346.534,Z 309.141,A -85,B 0,C 180,E1 14595.909,E2 14595.909} C_VEL
LIN {X 0,Y 343.963,Z 304.878,A -85,B 0,C 180,E1 14594.306,E2 14594.306} C_VEL
LIN {X 0,Y 340.972,Z 300.072,A -85,B 0,C 180,E1 14592.361,E2 14592.361} C_VEL
LIN {X 0,Y 337.486,Z 294.64,A -85,B 0,C 180,E1 14589.895,E2 14589.895} C_VEL
LIN {X 0,Y 334.803,Z 290.162,A -85,B 0,C 180,E1 14587.724,E2 14587.724} C_VEL
LIN {X 0,Y 331.709,Z 285.999,A -85,B 0,C 180,E1 14585.189,E2 14585.189} C_VEL
LIN {X 0,Y 330.739,Z 283.986,A -85,B 0,C 180,E1 14584.161,E2 14584.161} C_VEL
LIN {X 0,Y 327.976,Z 280.662,A -85,B 0,C 180,E1 14581.573,E2 14581.573} C_VEL
LIN {X 0,Y 326.796,Z 278.117,A -85,B 0,C 180,E1 14580.001,E2 14580.001} C_VEL
LIN {X 0,Y 323.941,Z 274.915,A -85,B 0,C 180,E1 14576.639,E2 14576.639} C_VEL
LIN {X 0,Y 322.694,Z 272.187,A -85,B 0,C 180,E1 14574.31,E2 14574.31} C_VEL
LIN {X 0,Y 319.171,Z 267.798,A -85,B 0,C 180,E1 14566.043,E2 14566.043} C_VEL
LIN {X 0,Y 318.746,Z 266.767,A -85,B 0,C 180,E1 14562.286,E2 14562.286} C_VEL
LIN {X 0,Y 318.829,Z 266.931,A -85,B 0,C 180,E1 14558.282,E2 14558.282} C_VEL
LIN {X 0,Y 319.455,Z 268.622,A -85,B 0,C 180,E1 14554.013,E2 14554.013} C_VEL
LIN {X 0,Y 322.873,Z 272.506,A -85,B 0,C 180,E1 14546.975,E2 14546.975} C_VEL
LIN {X 0,Y 325.413,Z 277.083,A -85,B 0,C 180,E1 14542.972,E2 14542.972} C_VEL
LIN {X 0,Y 326.893,Z 278.569,A -85,B 0,C 180,E1 14541.395,E2 14541.395} C_VEL
LIN {X 0,Y 328.905,Z 282.452,A -85,B 0,C 180,E1 14538.932,E2 14538.932} C_VEL
LIN {X 0,Y 330.483,Z 284.083,A -85,B 0,C 180,E1 14537.573,E2 14537.573} C_VEL
LIN {X 0,Y 332.582,Z 288.087,A -85,B 0,C 180,E1 14535.441,E2 14535.441} C_VEL
LIN {X 0,Y 334.003,Z 289.895,A -85,B 0,C 180,E1 14534.32,E2 14534.32} C_VEL
LIN {X 0,Y 336.474,Z 294.042,A -85,B 0,C 180,E1 14532.277,E2 14532.277} C_VEL
LIN {X 0,Y 337.755,Z 296.38,A -85,B 0,C 180,E1 14531.245,E2 14531.245} C_VEL
LIN {X 0,Y 340.353,Z 300.509,A -85,B 0,C 180,E1 14529.388,E2 14529.388} C_VEL
LIN {X 0,Y 343.912,Z 306.906,A -85,B 0,C 180,E1 14526.918,E2 14526.918} C_VEL
LIN {X 0,Y 348.258,Z 314.475,A -85,B 0,C 180,E1 14524.225,E2 14524.225} C_VEL
LIN {X 0,Y 354.67,Z 326.741,A -85,B 0,C 180,E1 14520.495,E2 14520.495} C_VEL
LIN {X 0,Y 361.128,Z 340.258,A -85,B 0,C 180,E1 14517.006,E2 14517.006} C_VEL
LIN {X 0,Y 367.474,Z 354.888,A -85,B 0,C 180,E1 14513.748,E2 14513.748} C_VEL
LIN {X 0,Y 369.757,Z 360.734,A -85,B 0,C 180,E1 14512.582,E2 14512.582} C_VEL
LIN {X 0,Y 364.225,Z 392.318,A -85,B 0,C 180,E1 14509.971,E2 14509.971} C_VEL
LIN {X 0,Y 368.525,Z 458.11,A -85,B 0,C 180,E1 14507.048,E2 14507.048} C_VEL
LIN {X 0,Y 358.32,Z 630.247,A -85,B 0,C 180,E1 14503.331,E2 14503.331} C_VEL
LIN {X 0,Y 356.384,Z 651.329,A -85,B 0,C 180,E1 14502.688,E2 14502.688} C_VEL
LIN {X 0,Y 353.776,Z 671.594,A -85,B 0,C 180,E1 14501.784,E2 14501.784} C_VEL
LIN {X 0,Y 350.581,Z 691.136,A -85,B 0,C 180,E1 14500.611,E2 14500.611} C_VEL
LIN {X 0,Y 346.942,Z 709.703,A -85,B 0,C 180,E1 14499.179,E2 14499.179} C_VEL
LIN {X 0,Y 343.065,Z 726.825,A -85,B 0,C 180,E1 14497.538,E2 14497.538} C_VEL
LIN {X 0,Y 338.899,Z 743.367,A -85,B 0,C 180,E1 14495.589,E2 14495.589} C_VEL
LIN {X 0,Y 334.763,Z 758.457,A -85,B 0,C 180,E1 14493.426,E2 14493.426} C_VEL
LIN {X 0,Y 330.767,Z 772.205,A -85,B 0,C 180,E1 14491.041,E2 14491.041} C_VEL
LIN {X 0,Y 326.741,Z 785.422,A -85,B 0,C 180,E1 14488.248,E2 14488.248} C_VEL
LIN {X 0,Y 323.098,Z 797.24,A -85,B 0,C 180,E1 14485.165,E2 14485.165} C_VEL
LIN {X 0,Y 320.075,Z 807.207,A -85,B 0,C 180,E1 14481.921,E2 14481.921} C_VEL
LIN {X 0,Y 318.234,Z 813.42,A -85,B 0,C 180,E1 14479.414,E2 14479.414} C_VEL
LIN {X 0,Y 316.492,Z 816.404,A -85,B 0,C 180,E1 14478.155,E2 14478.155} C_VEL
LIN {X 0,Y 308.9,Z 823.521,A -85,B 0,C 180,E1 14474.873,E2 14474.873} C_VEL
LIN {X 0,Y 307.604,Z 825.466,A -85,B 0,C 180,E1 14473.606,E2 14473.606} C_VEL
LIN {X 0,Y 306.709,Z 829.423,A -85,B 0,C 180,E1 14469.859,E2 14469.859} C_VEL
LIN {X 0,Y 306.331,Z 831.621,A -85,B 0,C 180,E1 14466.128,E2 14466.128} C_VEL
LIN {X 0,Y 306.348,Z 832.16,A -85,B 0,C 180,E1 14462.59,E2 14462.59} C_VEL
LIN {X 0,Y 306.74,Z 831.205,A -85,B 0,C 180,E1 14459.004,E2 14459.004} C_VEL
LIN {X 0,Y 307.631,Z 828.601,A -85,B 0,C 180,E1 14455.313,E2 14455.313} C_VEL
LIN {X 0,Y 309.166,Z 824.249,A -85,B 0,C 180,E1 14451.618,E2 14451.618} C_VEL
LIN {X 0,Y 311.347,Z 818.327,A -85,B 0,C 180,E1 14448.093,E2 14448.093} C_VEL
LIN {X 0,Y 314.296,Z 810.692,A -85,B 0,C 180,E1 14444.671,E2 14444.671} C_VEL
LIN {X 0,Y 317.795,Z 801.755,A -85,B 0,C 180,E1 14441.517,E2 14441.517} C_VEL
LIN {X 0,Y 322.131,Z 790.575,A -85,B 0,C 180,E1 14438.372,E2 14438.372} C_VEL
LIN {X 0,Y 327.031,Z 777.589,A -85,B 0,C 180,E1 14435.437,E2 14435.437} C_VEL
LIN {X 0,Y 332.169,Z 763.231,A -85,B 0,C 180,E1 14432.806,E2 14432.806} C_VEL
LIN {X 0,Y 337.457,Z 747.299,A -85,B 0,C 180,E1 14430.439,E2 14430.439} C_VEL
LIN {X 0,Y 342.599,Z 730.367,A -85,B 0,C 180,E1 14428.404,E2 14428.404} C_VEL
LIN {X 0,Y 347.366,Z 712.608,A -85,B 0,C 180,E1 14426.681,E2 14426.681} C_VEL
LIN {X 0,Y 351.679,Z 694.014,A -85,B 0,C 180,E1 14425.243,E2 14425.243} C_VEL
LIN {X 0,Y 355.255,Z 675.565,A -85,B 0,C 180,E1 14424.124,E2 14424.124} C_VEL
LIN {X 0,Y 358.405,Z 655.245,A -85,B 0,C 180,E1 14423.193,E2 14423.193} C_VEL
LIN {X 0,Y 360.803,Z 634.022,A -85,B 0,C 180,E1 14422.518,E2 14422.518} C_VEL
LIN {X 0,Y 372.487,Z 479.723,A -85,B 0,C 180,E1 14419.064,E2 14419.064} C_VEL
LIN {X 0,Y 373.773,Z 460.871,A -85,B 0,C 180,E1 14418.628,E2 14418.628} C_VEL
LIN {X 0,Y 371.951,Z 408.852,A -85,B 0,C 180,E1 14416.053,E2 14416.053} C_VEL
LIN {X 0,Y 370.935,Z 380.746,A -85,B 0,C 180,E1 14414.517,E2 14414.517} C_VEL
LIN {X 0,Y 372.594,Z 372.958,A -85,B 0,C 180,E1 14413.817,E2 14413.817} C_VEL
LIN {X 0,Y 368.656,Z 361.888,A -85,B 0,C 180,E1 14410.943,E2 14410.943} C_VEL
LIN {X 0,Y 365.244,Z 352.95,A -85,B 0,C 180,E1 14408.183,E2 14408.183} C_VEL
LIN {X 0,Y 362.043,Z 345.221,A -85,B 0,C 180,E1 14405.228,E2 14405.228} C_VEL
LIN {X 0,Y 360.125,Z 340.902,A -85,B 0,C 180,E1 14403.183,E2 14403.183} C_VEL
LIN {X 0,Y 358.669,Z 337.454,A -85,B 0,C 180,E1 14401.277,E2 14401.277} C_VEL
LIN {X 0,Y 357.187,Z 333.736,A -85,B 0,C 180,E1 14398.716,E2 14398.716} C_VEL
LIN {X 0,Y 355.72,Z 329.552,A -85,B 0,C 180,E1 14393.706,E2 14393.706} C_VEL
LIN {X 0,Y 355.957,Z 329.648,A -85,B 0,C 180,E1 14389.152,E2 14389.152} C_VEL
LIN {X 0,Y 356.336,Z 330.874,A -85,B 0,C 180,E1 14387.522,E2 14387.522} C_VEL
LIN {X 0,Y 358.611,Z 334.96,A -85,B 0,C 180,E1 14383.477,E2 14383.477} C_VEL
LIN {X 0,Y 361.026,Z 339.868,A -85,B 0,C 180,E1 14380.589,E2 14380.589} C_VEL
LIN {X 0,Y 363.419,Z 344.677,A -85,B 0,C 180,E1 14378.366,E2 14378.366} C_VEL
LIN {X 0,Y 365.305,Z 348.19,A -85,B 0,C 180,E1 14377.001,E2 14377.001} C_VEL
LIN {X 0,Y 373.001,Z 358.726,A -85,B 0,C 180,E1 14374.134,E2 14374.134} C_VEL
LIN {X 0,Y 380.746,Z 370.632,A -85,B 0,C 180,E1 14371.663,E2 14371.663} C_VEL
LIN {X 0,Y 382.87,Z 374.512,A -85,B 0,C 180,E1 14371.023,E2 14371.023} C_VEL
LIN {X 0,Y 373.53,Z 552.227,A -85,B 0,C 180,E1 14367.457,E2 14367.457} C_VEL
LIN {X 0,Y 368.67,Z 656.691,A -85,B 0,C 180,E1 14365.411,E2 14365.411} C_VEL
LIN {X 0,Y 366.314,Z 678.848,A -85,B 0,C 180,E1 14364.779,E2 14364.779} C_VEL
LIN {X 0,Y 362.894,Z 701.579,A -85,B 0,C 180,E1 14363.888,E2 14363.888} C_VEL
LIN {X 0,Y 359.053,Z 722.203,A -85,B 0,C 180,E1 14362.822,E2 14362.822} C_VEL
LIN {X 0,Y 354.513,Z 742.309,A -85,B 0,C 180,E1 14361.501,E2 14361.501} C_VEL
LIN {X 0,Y 349.585,Z 761.787,A -85,B 0,C 180,E1 14359.944,E2 14359.944} C_VEL
LIN {X 0,Y 344.089,Z 781.088,A -85,B 0,C 180,E1 14358.06,E2 14358.06} C_VEL
LIN {X 0,Y 337.977,Z 800.998,A -85,B 0,C 180,E1 14355.716,E2 14355.716} C_VEL
LIN {X 0,Y 332.048,Z 819.4,A -85,B 0,C 180,E1 14353.118,E2 14353.118} C_VEL
LIN {X 0,Y 326.407,Z 836.25,A -85,B 0,C 180,E1 14350.263,E2 14350.263} C_VEL
LIN {X 0,Y 320.932,Z 852.688,A -85,B 0,C 180,E1 14346.959,E2 14346.959} C_VEL
LIN {X 0,Y 316.358,Z 866.989,A -85,B 0,C 180,E1 14343.577,E2 14343.577} C_VEL
LIN {X 0,Y 312.38,Z 880.164,A -85,B 0,C 180,E1 14339.84,E2 14339.84} C_VEL
LIN {X 0,Y 309.105,Z 892.496,A -85,B 0,C 180,E1 14335.684,E2 14335.684} C_VEL
LIN {X 0,Y 306.922,Z 902.584,A -85,B 0,C 180,E1 14331.597,E2 14331.597} C_VEL
LIN {X 0,Y 305.611,Z 910.674,A -85,B 0,C 180,E1 14327.515,E2 14327.515} C_VEL
LIN {X 0,Y 304.968,Z 917.165,A -85,B 0,C 180,E1 14323.459,E2 14323.459} C_VEL
LIN {X 0,Y 304.799,Z 921.659,A -85,B 0,C 180,E1 14319.629,E2 14319.629} C_VEL
LIN {X 0,Y 304.883,Z 924.652,A -85,B 0,C 180,E1 14316.022,E2 14316.022} C_VEL
LIN {X 0,Y 304.969,Z 926.333,A -85,B 0,C 180,E1 14312.253,E2 14312.253} C_VEL
LIN {X 0,Y 304.976,Z 926.558,A -85,B 0,C 180,E1 14308.871,E2 14308.871} C_VEL
LIN {X 0,Y 304.9,Z 925.707,A -85,B 0,C 180,E1 14305.673,E2 14305.673} C_VEL
LIN {X 0,Y 304.779,Z 923.407,A -85,B 0,C 180,E1 14301.889,E2 14301.889} C_VEL
LIN {X 0,Y 304.831,Z 919.491,A -85,B 0,C 180,E1 14298.072,E2 14298.072} C_VEL
LIN {X 0,Y 305.188,Z 914.47,A -85,B 0,C 180,E1 14294.41,E2 14294.41} C_VEL
LIN {X 0,Y 306.17,Z 907.248,A -85,B 0,C 180,E1 14290.343,E2 14290.343} C_VEL
LIN {X 0,Y 307.848,Z 898.767,A -85,B 0,C 180,E1 14286.452,E2 14286.452} C_VEL
LIN {X 0,Y 310.379,Z 888.416,A -85,B 0,C 180,E1 14282.568,E2 14282.568} C_VEL
LIN {X 0,Y 313.658,Z 876.91,A -85,B 0,C 180,E1 14278.906,E2 14278.906} C_VEL
LIN {X 0,Y 317.865,Z 863.263,A -85,B 0,C 180,E1 14275.294,E2 14275.294} C_VEL
LIN {X 0,Y 323.054,Z 847.367,A -85,B 0,C 180,E1 14271.755,E2 14271.755} C_VEL
LIN {X 0,Y 328.318,Z 831.555,A -85,B 0,C 180,E1 14268.783,E2 14268.783} C_VEL
LIN {X 0,Y 333.817,Z 814.465,A -85,B 0,C 180,E1 14266.099,E2 14266.099} C_VEL
LIN {X 0,Y 339.932,Z 794.917,A -85,B 0,C 180,E1 14263.526,E2 14263.526} C_VEL
LIN {X 0,Y 345.478,Z 775.933,A -85,B 0,C 180,E1 14261.444,E2 14261.444} C_VEL
LIN {X 0,Y 350.669,Z 756.07,A -85,B 0,C 180,E1 14259.658,E2 14259.658} C_VEL
LIN {X 0,Y 355.679,Z 734.676,A -85,B 0,C 180,E1 14258.081,E2 14258.081} C_VEL
LIN {X 0,Y 359.874,Z 713.879,A -85,B 0,C 180,E1 14256.852,E2 14256.852} C_VEL
LIN {X 0,Y 363.439,Z 691.944,A -85,B 0,C 180,E1 14255.853,E2 14255.853} C_VEL
LIN {X 0,Y 366.326,Z 669.262,A -85,B 0,C 180,E1 14255.09,E2 14255.09} C_VEL
LIN {X 0,Y 367.98,Z 647.516,A -85,B 0,C 180,E1 14254.569,E2 14254.569} C_VEL
LIN {X 0,Y 376.672,Z 455.707,A -85,B 0,C 180,E1 14250.825,E2 14250.825} C_VEL
LIN {X 0,Y 380.641,Z 374.323,A -85,B 0,C 180,E1 14249.183,E2 14249.183} C_VEL
LIN {X 0,Y 369.333,Z 357.368,A -85,B 0,C 180,E1 14246.445,E2 14246.445} C_VEL
LIN {X 0,Y 357.208,Z 340.62,A -85,B 0,C 180,E1 14243.202,E2 14243.202} C_VEL
LIN {X 0,Y 354.75,Z 337.11,A -85,B 0,C 180,E1 14242.365,E2 14242.365} C_VEL
LIN {X 0,Y 348.201,Z 325.457,A -85,B 0,C 180,E1 14238.934,E2 14238.934} C_VEL
LIN {X 0,Y 342.674,Z 316.12,A -85,B 0,C 180,E1 14235.745,E2 14235.745} C_VEL
LIN {X 0,Y 339.558,Z 311.073,A -85,B 0,C 180,E1 14233.799,E2 14233.799} C_VEL
LIN {X 0,Y 336.88,Z 306.687,A -85,B 0,C 180,E1 14231.992,E2 14231.992} C_VEL
LIN {X 0,Y 333.674,Z 301.546,A -85,B 0,C 180,E1 14229.661,E2 14229.661} C_VEL
LIN {X 0,Y 330.471,Z 296.413,A -85,B 0,C 180,E1 14227.068,E2 14227.068} C_VEL
LIN {X 0,Y 327.794,Z 292.499,A -85,B 0,C 180,E1 14224.725,E2 14224.725} C_VEL
LIN {X 0,Y 326.953,Z 290.933,A -85,B 0,C 180,E1 14223.858,E2 14223.858} C_VEL
LIN {X 0,Y 324.282,Z 287.505,A -85,B 0,C 180,E1 14221.237,E2 14221.237} C_VEL
LIN {X 0,Y 323.26,Z 285.249,A -85,B 0,C 180,E1 14219.823,E2 14219.823} C_VEL
LIN {X 0,Y 320.437,Z 282.004,A -85,B 0,C 180,E1 14216.423,E2 14216.423} C_VEL
LIN {X 0,Y 319.311,Z 279.433,A -85,B 0,C 180,E1 14214.25,E2 14214.25} C_VEL
LIN {X 0,Y 315.835,Z 275.106,A -85,B 0,C 180,E1 14206.079,E2 14206.079} C_VEL
LIN {X 0,Y 315.403,Z 274.035,A -85,B 0,C 180,E1 14202.283,E2 14202.283} C_VEL
LIN {X 0,Y 315.482,Z 274.206,A -85,B 0,C 180,E1 14198.222,E2 14198.222} C_VEL
LIN {X 0,Y 316.049,Z 275.838,A -85,B 0,C 180,E1 14194.115,E2 14194.115} C_VEL
LIN {X 0,Y 319.404,Z 279.774,A -85,B 0,C 180,E1 14186.998,E2 14186.998} C_VEL
LIN {X 0,Y 321.771,Z 284.151,A -85,B 0,C 180,E1 14183.151,E2 14183.151} C_VEL
LIN {X 0,Y 323.227,Z 285.682,A -85,B 0,C 180,E1 14181.556,E2 14181.556} C_VEL
LIN {X 0,Y 325.424,Z 289.735,A -85,B 0,C 180,E1 14178.891,E2 14178.891} C_VEL
LIN {X 0,Y 326.734,Z 291.297,A -85,B 0,C 180,E1 14177.684,E2 14177.684} C_VEL
LIN {X 0,Y 329.179,Z 295.507,A -85,B 0,C 180,E1 14175.299,E2 14175.299} C_VEL
LIN {X 0,Y 330.226,Z 297.176,A -85,B 0,C 180,E1 14174.382,E2 14174.382} C_VEL
LIN {X 0,Y 333.223,Z 302.087,A -85,B 0,C 180,E1 14171.916,E2 14171.916} C_VEL
LIN {X 0,Y 336.49,Z 307.82,A -85,B 0,C 180,E1 14169.416,E2 14169.416} C_VEL
LIN {X 0,Y 339.781,Z 313.7,A -85,B 0,C 180,E1 14167.114,E2 14167.114} C_VEL
LIN {X 0,Y 343.763,Z 320.794,A -85,B 0,C 180,E1 14164.555,E2 14164.555} C_VEL
LIN {X 0,Y 349.98,Z 332.873,A -85,B 0,C 180,E1 14160.838,E2 14160.838} C_VEL
LIN {X 0,Y 356.293,Z 346.356,A -85,B 0,C 180,E1 14157.313,E2 14157.313} C_VEL
LIN {X 0,Y 362.421,Z 360.809,A -85,B 0,C 180,E1 14154.055,E2 14154.055} C_VEL
LIN {X 0,Y 363.876,Z 364.703,A -85,B 0,C 180,E1 14153.267,E2 14153.267} C_VEL
LIN {X 0,Y 359.045,Z 391.45,A -85,B 0,C 180,E1 14151.044,E2 14151.044} C_VEL
LIN {X 0,Y 363.19,Z 459.224,A -85,B 0,C 180,E1 14147.971,E2 14147.971} C_VEL
LIN {X 0,Y 352.616,Z 630.808,A -85,B 0,C 180,E1 14144.231,E2 14144.231} C_VEL
LIN {X 0,Y 350.579,Z 652.082,A -85,B 0,C 180,E1 14143.573,E2 14143.573} C_VEL
LIN {X 0,Y 347.769,Z 672.965,A -85,B 0,C 180,E1 14142.623,E2 14142.623} C_VEL
LIN {X 0,Y 344.331,Z 693.012,A -85,B 0,C 180,E1 14141.39,E2 14141.39} C_VEL
LIN {X 0,Y 340.445,Z 711.874,A -85,B 0,C 180,E1 14139.895,E2 14139.895} C_VEL
LIN {X 0,Y 336.184,Z 729.727,A -85,B 0,C 180,E1 14138.123,E2 14138.123} C_VEL
LIN {X 0,Y 331.711,Z 746.552,A -85,B 0,C 180,E1 14136.058,E2 14136.058} C_VEL
LIN {X 0,Y 327.136,Z 762.315,A -85,B 0,C 180,E1 14133.682,E2 14133.682} C_VEL
LIN {X 0,Y 322.765,Z 776.485,A -85,B 0,C 180,E1 14131.067,E2 14131.067} C_VEL
LIN {X 0,Y 318.694,Z 789.165,A -85,B 0,C 180,E1 14128.204,E2 14128.204} C_VEL
LIN {X 0,Y 315.073,Z 800.366,A -85,B 0,C 180,E1 14125.087,E2 14125.087} C_VEL
LIN {X 0,Y 311.981,Z 810.074,A -85,B 0,C 180,E1 14121.71,E2 14121.71} C_VEL
LIN {X 0,Y 309.566,Z 818.089,A -85,B 0,C 180,E1 14118.134,E2 14118.134} C_VEL
LIN {X 0,Y 307.927,Z 824.112,A -85,B 0,C 180,E1 14114.56,E2 14114.56} C_VEL
LIN {X 0,Y 307.604,Z 825.466,A -85,B 0,C 180,E1 14113.606,E2 14113.606} C_VEL
LIN {X 0,Y 306.23,Z 827.422,A -85,B 0,C 180,E1 14112.227,E2 14112.227} C_VEL
LIN {X 0,Y 300.934,Z 830.741,A -85,B 0,C 180,E1 14109.51,E2 14109.51} C_VEL
LIN {X 0,Y 298.679,Z 832.12,A -85,B 0,C 180,E1 14107.766,E2 14107.766} C_VEL
LIN {X 0,Y 298.49,Z 832.373,A -85,B 0,C 180,E1 14107.234,E2 14107.234} C_VEL
LIN {X 0,Y 298.413,Z 833.406,A -85,B 0,C 180,E1 14103.455,E2 14103.455} C_VEL
LIN {X 0,Y 298.739,Z 832.865,A -85,B 0,C 180,E1 14099.71,E2 14099.71} C_VEL
LIN {X 0,Y 299.582,Z 830.63,A -85,B 0,C 180,E1 14095.861,E2 14095.861} C_VEL
LIN {X 0,Y 301.157,Z 826.454,A -85,B 0,C 180,E1 14091.891,E2 14091.891} C_VEL
LIN {X 0,Y 303.512,Z 820.442,A -85,B 0,C 180,E1 14088.033,E2 14088.033} C_VEL
LIN {X 0,Y 306.634,Z 812.831,A -85,B 0,C 180,E1 14084.433,E2 14084.433} C_VEL
LIN {X 0,Y 310.406,Z 803.683,A -85,B 0,C 180,E1 14081.079,E2 14081.079} C_VEL
LIN {X 0,Y 314.869,Z 792.819,A -85,B 0,C 180,E1 14077.902,E2 14077.902} C_VEL
LIN {X 0,Y 319.786,Z 780.503,A -85,B 0,C 180,E1 14075.001,E2 14075.001} C_VEL
LIN {X 0,Y 324.743,Z 767.405,A -85,B 0,C 180,E1 14072.479,E2 14072.479} C_VEL
LIN {X 0,Y 330.009,Z 752.627,A -85,B 0,C 180,E1 14070.139,E2 14070.139} C_VEL
LIN {X 0,Y 335.303,Z 736.395,A -85,B 0,C 180,E1 14068.04,E2 14068.04} C_VEL
LIN {X 0,Y 340.464,Z 718.727,A -85,B 0,C 180,E1 14066.197,E2 14066.197} C_VEL
LIN {X 0,Y 345.144,Z 700.306,A -85,B 0,C 180,E1 14064.654,E2 14064.654} C_VEL
LIN {X 0,Y 349.165,Z 681.68,A -85,B 0,C 180,E1 14063.424,E2 14063.424} C_VEL
LIN {X 0,Y 352.67,Z 661.574,A -85,B 0,C 180,E1 14062.413,E2 14062.413} C_VEL
LIN {X 0,Y 355.415,Z 640.43,A -85,B 0,C 180,E1 14061.659,E2 14061.659} C_VEL
LIN {X 0,Y 365.784,Z 509.934,A -85,B 0,C 180,E1 14058.678,E2 14058.678} C_VEL
LIN {X 0,Y 369.369,Z 462.312,A -85,B 0,C 180,E1 14057.617,E2 14057.617} C_VEL
LIN {X 0,Y 367.901,Z 410.57,A -85,B 0,C 180,E1 14055.012,E2 14055.012} C_VEL
LIN {X 0,Y 367.073,Z 379.419,A -85,B 0,C 180,E1 14053.266,E2 14053.266} C_VEL
LIN {X 0,Y 367.371,Z 377.385,A -85,B 0,C 180,E1 14053.055,E2 14053.055} C_VEL
LIN {X 0,Y 363.46,Z 366.023,A -85,B 0,C 180,E1 14049.98,E2 14049.98} C_VEL
LIN {X 0,Y 359.806,Z 356.246,A -85,B 0,C 180,E1 14046.702,E2 14046.702} C_VEL
LIN {X 0,Y 356.86,Z 348.789,A -85,B 0,C 180,E1 14043.533,E2 14043.533} C_VEL
LIN {X 0,Y 354.887,Z 344.291,A -85,B 0,C 180,E1 14040.968,E2 14040.968} C_VEL
LIN {X 0,Y 353.626,Z 340.84,A -85,B 0,C 180,E1 14038.541,E2 14038.541} C_VEL
LIN {X 0,Y 352.325,Z 336.791,A -85,B 0,C 180,E1 14033.645,E2 14033.645} C_VEL
LIN {X 0,Y 352.65,Z 336.947,A -85,B 0,C 180,E1 14029.049,E2 14029.049} C_VEL
LIN {X 0,Y 355.018,Z 341.812,A -85,B 0,C 180,E1 14023.809,E2 14023.809} C_VEL
LIN {X 0,Y 357.313,Z 346.7,A -85,B 0,C 180,E1 14020.889,E2 14020.889} C_VEL
LIN {X 0,Y 359.284,Z 350.285,A -85,B 0,C 180,E1 14019.174,E2 14019.174} C_VEL
LIN {X 0,Y 365.301,Z 358.34,A -85,B 0,C 180,E1 14016.531,E2 14016.531} C_VEL
LIN {X 0,Y 372.582,Z 368.97,A -85,B 0,C 180,E1 14013.846,E2 14013.846} C_VEL
LIN {X 0,Y 378.387,Z 378.566,A -85,B 0,C 180,E1 14011.966,E2 14011.966} C_VEL
LIN {X 0,Y 368.776,Z 551.75,A -85,B 0,C 180,E1 14008.462,E2 14008.462} C_VEL
LIN {X 0,Y 363.595,Z 656.633,A -85,B 0,C 180,E1 14006.383,E2 14006.383} C_VEL
LIN {X 0,Y 361.146,Z 678.815,A -85,B 0,C 180,E1 14005.746,E2 14005.746} C_VEL
LIN {X 0,Y 357.753,Z 700.588,A -85,B 0,C 180,E1 14004.893,E2 14004.893} C_VEL
LIN {X 0,Y 353.816,Z 720.942,A -85,B 0,C 180,E1 14003.843,E2 14003.843} C_VEL
LIN {X 0,Y 349.062,Z 741.328,A -85,B 0,C 180,E1 14002.505,E2 14002.505} C_VEL
LIN {X 0,Y 343.882,Z 761.07,A -85,B 0,C 180,E1 14000.921,E2 14000.921} C_VEL
LIN {X 0,Y 338.235,Z 780.112,A -85,B 0,C 180,E1 13999.047,E2 13999.047} C_VEL
LIN {X 0,Y 331.86,Z 800.01,A -85,B 0,C 180,E1 13996.683,E2 13996.683} C_VEL
LIN {X 0,Y 325.839,Z 817.846,A -85,B 0,C 180,E1 13994.149,E2 13994.149} C_VEL
LIN {X 0,Y 319.743,Z 835.219,A -85,B 0,C 180,E1 13991.163,E2 13991.163} C_VEL
LIN {X 0,Y 314.04,Z 851.438,A -85,B 0,C 180,E1 13987.852,E2 13987.852} C_VEL
LIN {X 0,Y 309.269,Z 865.544,A -85,B 0,C 180,E1 13984.453,E2 13984.453} C_VEL
LIN {X 0,Y 305.115,Z 878.425,A -85,B 0,C 180,E1 13980.742,E2 13980.742} C_VEL
LIN {X 0,Y 301.642,Z 890.608,A -85,B 0,C 180,E1 13976.58,E2 13976.58} C_VEL
LIN {X 0,Y 299.335,Z 900.329,A -85,B 0,C 180,E1 13972.587,E2 13972.587} C_VEL
LIN {X 0,Y 297.838,Z 908.669,A -85,B 0,C 180,E1 13968.392,E2 13968.392} C_VEL
LIN {X 0,Y 297.111,Z 915.037,A -85,B 0,C 180,E1 13964.418,E2 13964.418} C_VEL
LIN {X 0,Y 296.866,Z 920.024,A -85,B 0,C 180,E1 13960.281,E2 13960.281} C_VEL
LIN {X 0,Y 296.938,Z 923.113,A -85,B 0,C 180,E1 13956.619,E2 13956.619} C_VEL
LIN {X 0,Y 297.044,Z 925.04,A -85,B 0,C 180,E1 13952.699,E2 13952.699} C_VEL
LIN {X 0,Y 297.07,Z 925.357,A -85,B 0,C 180,E1 13949.034,E2 13949.034} C_VEL
LIN {X 0,Y 296.99,Z 924.553,A -85,B 0,C 180,E1 13945.75,E2 13945.75} C_VEL
LIN {X 0,Y 296.854,Z 922.399,A -85,B 0,C 180,E1 13941.993,E2 13941.993} C_VEL
LIN {X 0,Y 296.887,Z 918.448,A -85,B 0,C 180,E1 13937.946,E2 13937.946} C_VEL
LIN {X 0,Y 297.257,Z 913.419,A -85,B 0,C 180,E1 13934.154,E2 13934.154} C_VEL
LIN {X 0,Y 298.351,Z 905.902,A -85,B 0,C 180,E1 13929.805,E2 13929.805} C_VEL
LIN {X 0,Y 300.157,Z 897.367,A -85,B 0,C 180,E1 13925.81,E2 13925.81} C_VEL
LIN {X 0,Y 302.885,Z 886.892,A -85,B 0,C 180,E1 13921.812,E2 13921.812} C_VEL
LIN {X 0,Y 306.592,Z 874.666,A -85,B 0,C 180,E1 13917.886,E2 13917.886} C_VEL
LIN {X 0,Y 310.844,Z 861.621,A -85,B 0,C 180,E1 13914.392,E2 13914.392} C_VEL
LIN {X 0,Y 316.03,Z 846.496,A -85,B 0,C 180,E1 13910.978,E2 13910.978} C_VEL
LIN {X 0,Y 321.573,Z 830.553,A -85,B 0,C 180,E1 13907.927,E2 13907.927} C_VEL
LIN {X 0,Y 327.312,Z 813.484,A -85,B 0,C 180,E1 13905.215,E2 13905.215} C_VEL
LIN {X 0,Y 333.574,Z 794.118,A -85,B 0,C 180,E1 13902.642,E2 13902.642} C_VEL
LIN {X 0,Y 339.373,Z 774.981,A -85,B 0,C 180,E1 13900.524,E2 13900.524} C_VEL
LIN {X 0,Y 344.752,Z 755.094,A -85,B 0,C 180,E1 13898.723,E2 13898.723} C_VEL
LIN {X 0,Y 349.938,Z 733.604,A -85,B 0,C 180,E1 13897.137,E2 13897.137} C_VEL
LIN {X 0,Y 354.274,Z 712.668,A -85,B 0,C 180,E1 13895.903,E2 13895.903} C_VEL
LIN {X 0,Y 357.919,Z 690.61,A -85,B 0,C 180,E1 13894.908,E2 13894.908} C_VEL
LIN {X 0,Y 360.953,Z 666.643,A -85,B 0,C 180,E1 13894.123,E2 13894.123} C_VEL
LIN {X 0,Y 362.608,Z 644.022,A -85,B 0,C 180,E1 13893.59,E2 13893.59} C_VEL
LIN {X 0,Y 371.295,Z 459.919,A -85,B 0,C 180,E1 13889.97,E2 13889.97} C_VEL
LIN {X 0,Y 375.47,Z 378.169,A -85,B 0,C 180,E1 13888.317,E2 13888.317} C_VEL
LIN {X 0,Y 363.668,Z 360.568,A -85,B 0,C 180,E1 13885.355,E2 13885.355} C_VEL
LIN {X 0,Y 352.868,Z 345.767,A -85,B 0,C 180,E1 13882.359,E2 13882.359} C_VEL
LIN {X 0,Y 348.057,Z 339.333,A -85,B 0,C 180,E1 13880.868,E2 13880.868} C_VEL
LIN {X 0,Y 342.078,Z 328.54,A -85,B 0,C 180,E1 13877.522,E2 13877.522} C_VEL
LIN {X 0,Y 336.255,Z 318.742,A -85,B 0,C 180,E1 13873.937,E2 13873.937} C_VEL
LIN {X 0,Y 332.653,Z 313.081,A -85,B 0,C 180,E1 13871.513,E2 13871.513} C_VEL
LIN {X 0,Y 329.624,Z 308.164,A -85,B 0,C 180,E1 13869.252,E2 13869.252} C_VEL
LIN {X 0,Y 326.753,Z 303.407,A -85,B 0,C 180,E1 13866.855,E2 13866.855} C_VEL
LIN {X 0,Y 324.036,Z 299.355,A -85,B 0,C 180,E1 13864.425,E2 13864.425} C_VEL
LIN {X 0,Y 323.179,Z 297.875,A -85,B 0,C 180,E1 13863.548,E2 13863.548} C_VEL
LIN {X 0,Y 320.6,Z 294.347,A -85,B 0,C 180,E1 13860.894,E2 13860.894} C_VEL
LIN {X 0,Y 319.721,Z 292.378,A -85,B 0,C 180,E1 13859.642,E2 13859.642} C_VEL
LIN {X 0,Y 316.941,Z 289.094,A -85,B 0,C 180,E1 13856.202,E2 13856.202} C_VEL
LIN {X 0,Y 315.806,Z 286.569,A -85,B 0,C 180,E1 13854.004,E2 13854.004} C_VEL
LIN {X 0,Y 312.418,Z 282.142,A -85,B 0,C 180,E1 13845.545,E2 13845.545} C_VEL
LIN {X 0,Y 312.058,Z 281.197,A -85,B 0,C 180,E1 13841.507,E2 13841.507} C_VEL
LIN {X 0,Y 312.229,Z 281.701,A -85,B 0,C 180,E1 13837.263,E2 13837.263} C_VEL
LIN {X 0,Y 313.701,Z 284.732,A -85,B 0,C 180,E1 13831.023,E2 13831.023} C_VEL
LIN {X 0,Y 315.93,Z 287.081,A -85,B 0,C 180,E1 13827.021,E2 13827.021} C_VEL
LIN {X 0,Y 318.217,Z 291.296,A -85,B 0,C 180,E1 13823.249,E2 13823.249} C_VEL
LIN {X 0,Y 319.566,Z 292.803,A -85,B 0,C 180,E1 13821.721,E2 13821.721} C_VEL
LIN {X 0,Y 321.753,Z 296.8,A -85,B 0,C 180,E1 13819.029,E2 13819.029} C_VEL
LIN {X 0,Y 322.842,Z 298.033,A -85,B 0,C 180,E1 13818.014,E2 13818.014} C_VEL
LIN {X 0,Y 325.357,Z 302.461,A -85,B 0,C 180,E1 13815.478,E2 13815.478} C_VEL
LIN {X 0,Y 326.436,Z 304.376,A -85,B 0,C 180,E1 13814.467,E2 13814.467} C_VEL
LIN {X 0,Y 329.192,Z 308.881,A -85,B 0,C 180,E1 13812.165,E2 13812.165} C_VEL
LIN {X 0,Y 332.449,Z 314.683,A -85,B 0,C 180,E1 13809.615,E2 13809.615} C_VEL
LIN {X 0,Y 337.038,Z 322.846,A -85,B 0,C 180,E1 13806.395,E2 13806.395} C_VEL
LIN {X 0,Y 343.317,Z 334.952,A -85,B 0,C 180,E1 13802.375,E2 13802.375} C_VEL
LIN {X 0,Y 349.688,Z 348.469,A -85,B 0,C 180,E1 13798.624,E2 13798.624} C_VEL
LIN {X 0,Y 355.406,Z 361.845,A -85,B 0,C 180,E1 13795.439,E2 13795.439} C_VEL
LIN {X 0,Y 358.065,Z 368.621,A -85,B 0,C 180,E1 13793.982,E2 13793.982} C_VEL
LIN {X 0,Y 353.963,Z 390.628,A -85,B 0,C 180,E1 13792.141,E2 13792.141} C_VEL
LIN {X 0,Y 357.945,Z 460.29,A -85,B 0,C 180,E1 13788.924,E2 13788.924} C_VEL
LIN {X 0,Y 347.037,Z 630.904,A -85,B 0,C 180,E1 13785.172,E2 13785.172} C_VEL
LIN {X 0,Y 344.945,Z 652.13,A -85,B 0,C 180,E1 13784.513,E2 13784.513} C_VEL
LIN {X 0,Y 342.1,Z 672.702,A -85,B 0,C 180,E1 13783.579,E2 13783.579} C_VEL
LIN {X 0,Y 338.608,Z 692.538,A -85,B 0,C 180,E1 13782.363,E2 13782.363} C_VEL
LIN {X 0,Y 334.559,Z 711.627,A -85,B 0,C 180,E1 13780.854,E2 13780.854} C_VEL
LIN {X 0,Y 330.039,Z 729.942,A -85,B 0,C 180,E1 13779.032,E2 13779.032} C_VEL
LIN {X 0,Y 325.253,Z 747.258,A -85,B 0,C 180,E1 13776.887,E2 13776.887} C_VEL
LIN {X 0,Y 320.472,Z 763.059,A -85,B 0,C 180,E1 13774.475,E2 13774.475} C_VEL
LIN {X 0,Y 315.891,Z 777.27,A -85,B 0,C 180,E1 13771.816,E2 13771.816} C_VEL
LIN {X 0,Y 311.61,Z 790.001,A -85,B 0,C 180,E1 13768.899,E2 13768.899} C_VEL
LIN {X 0,Y 307.787,Z 801.253,A -85,B 0,C 180,E1 13765.717,E2 13765.717} C_VEL
LIN {X 0,Y 304.511,Z 811.012,A -85,B 0,C 180,E1 13762.265,E2 13762.265} C_VEL
LIN {X 0,Y 302.012,Z 818.825,A -85,B 0,C 180,E1 13758.738,E2 13758.738} C_VEL
LIN {X 0,Y 300.253,Z 824.879,A -85,B 0,C 180,E1 13755.145,E2 13755.145} C_VEL
LIN {X 0,Y 299.127,Z 829.298,A -85,B 0,C 180,E1 13751.488,E2 13751.488} C_VEL
LIN {X 0,Y 298.542,Z 832.142,A -85,B 0,C 180,E1 13747.765,E2 13747.765} C_VEL
LIN {X 0,Y 298.49,Z 832.373,A -85,B 0,C 180,E1 13747.234,E2 13747.234} C_VEL
LIN {X 0,Y 297.415,Z 833.157,A -85,B 0,C 180,E1 13745.762,E2 13745.762} C_VEL
LIN {X 0,Y 292.364,Z 834.385,A -85,B 0,C 180,E1 13742.654,E2 13742.654} C_VEL
LIN {X 0,Y 290.768,Z 834.441,A -85,B 0,C 180,E1 13740.926,E2 13740.926} C_VEL
LIN {X 0,Y 290.739,Z 834.351,A -85,B 0,C 180,E1 13740.486,E2 13740.486} C_VEL
LIN {X 0,Y 291.502,Z 832.494,A -85,B 0,C 180,E1 13736.483,E2 13736.483} C_VEL
LIN {X 0,Y 292.925,Z 828.977,A -85,B 0,C 180,E1 13732.589,E2 13732.589} C_VEL
LIN {X 0,Y 295.163,Z 823.59,A -85,B 0,C 180,E1 13728.661,E2 13728.661} C_VEL
LIN {X 0,Y 298.18,Z 816.621,A -85,B 0,C 180,E1 13724.97,E2 13724.97} C_VEL
LIN {X 0,Y 301.973,Z 808.026,A -85,B 0,C 180,E1 13721.468,E2 13721.468} C_VEL
LIN {X 0,Y 306.197,Z 798.415,A -85,B 0,C 180,E1 13718.346,E2 13718.346} C_VEL
LIN {X 0,Y 311.377,Z 786.314,A -85,B 0,C 180,E1 13715.197,E2 13715.197} C_VEL
LIN {X 0,Y 316.68,Z 773.348,A -85,B 0,C 180,E1 13712.461,E2 13712.461} C_VEL
